	_InputStopController : MockPluginAutomationController(name := "InputController");
	_InputStopBranch : MockCompositeAutomationComponent(name := "InputBranch", parent := _InputStopController);

	_LifecycleLeaf : MockLeafAutomationComponent(name := "TestLeaf", parent := _TimeoutRoot);
	_EnableDisableLeaf : MockLeafAutomationComponent(name := "EnDisLeaf", parent := _TimeoutRoot);
	_IgnoreComposite : MockCompositeAutomationComponent(name := "CompIgnore", parent := _TimeoutRoot);
	_ContinueComposite : MockCompositeAutomationComponent(name := "CompContinue", parent := _TimeoutRoot);
	_StopComposite : MockCompositeAutomationComponent(name := "CompStop", parent := _TimeoutRoot);
	_BubbleComposite : MockCompositeAutomationComponent(name := "CompBubble", parent := _TimeoutRoot);
	_BubbleEvent : MockAutomationEvent(sourceObject := 0, eventId := 10, payload := "BubblePayload");
	_StopBubbleComposite : MockCompositeAutomationComponent(name := "CompStopBubble", parent := _TimeoutRoot);
	_StopBubbleEvent : MockAutomationEvent(sourceObject := 0, eventId := 20, payload := "StopPayload");
	_BroadcastComposite : MockCompositeAutomationComponent(name := "CompBcast", parent := _TimeoutRoot);
	_BroadcastEvent : MockAutomationEvent(sourceObject := 0, eventId := 30, payload := "BcastPayload");
	_InputOutputLeaf : MockLeafAutomationComponent(name := "IOLeaf", parent := _TimeoutRoot);
	_OutputPoliciesBranch : MockCompositeAutomationComponent(name := "OutputPolicies", parent := _TimeoutRoot);
	_InitializingProbeLeaf : MockLeafAutomationComponent(name := "InitProbe", parent := _TimeoutRoot);
	_WorkingProbeLeaf : MockLeafAutomationComponent(name := "WorkProbe", parent := _TimeoutRoot);
	_CallbackResetComposite : MockCompositeAutomationComponent(name := "CallbackReset", parent := _TimeoutRoot);
	_DuplicateBranch : MockCompositeAutomationComponent(name := "Duplicate", parent := _TimeoutRoot);
	_WrongParentBranch : MockCompositeAutomationComponent(name := "WrongParent", parent := _TimeoutRoot);
	_ForeignChildLeaf : MockLeafAutomationComponent(name := "Foreign", parent := _TimeoutRoot);

	_ResetPolicyLeaf : MockLeafAutomationComponent(name := "ResetPolicyLeaf", parent := _TimeoutRoot);
	_BeforeResetPolicyBranch : MockCompositeAutomationComponent(name := "BeforeResetPolicy", parent := _TimeoutRoot);
	_AfterResetPolicyBranch : MockCompositeAutomationComponent(name := "AfterResetPolicy", parent := _TimeoutRoot);
	_RecoverPolicyLeaf : MockLeafAutomationComponent(name := "RecoverPolicyLeaf", parent := _TimeoutRoot);
	_RecoverPolicyBranch : MockCompositeAutomationComponent(name := "RecoverPolicyBranch", parent := _TimeoutRoot);

	_AfterInitBranch : MockCompositeAutomationComponent(name := "AfterInitBranch", parent := _TimeoutRoot);
	_TimeoutNormLeaf : MockLeafAutomationComponent(name := "TimeoutNormLeaf", parent := _TimeoutRoot);

	_DisabledChildBranch : MockCompositeAutomationComponent(name := "DisabledChildBranch", parent := _TimeoutRoot);
	_CmdHmiPlugin : MockHmiControllerPlugin;
	_CmdHmiPlugins : ARRAY [0..0] OF TOF_Automation.IAutomationControllerPlugin := [_CmdHmiPlugin];
	_CmdHmiController : MockPluginAutomationController(name := "CmdHmiController");
END_VAR

(*!
<summary>Dispatches one scenario against the fresh fixture.</summary>
<description>Call once per fixture. Each method uses the assertions of the receiving case.</description>
<param name="scenario">Scenario assigned to the caller.</param>
<param name="assertions">Valid assertion context borrowed from the active case.</param>
*)
METHOD ExecuteScenario
VAR_INPUT
	scenario : AUTOMATION_COMPONENT_TEST_SCENARIO;
	assertions : REFERENCE TO TOF_Testing.Assertions;
END_VAR
CASE scenario OF
	AUTOMATION_COMPONENT_TEST_SCENARIO.LIFECYCLE_TRANSITIONS:
		testLifecycleTransitions(assertions := assertions);

	AUTOMATION_COMPONENT_TEST_SCENARIO.ENABLE_DISABLE:
		testEnableDisable(assertions := assertions);

	AUTOMATION_COMPONENT_TEST_SCENARIO.CHILD_ERROR_POLICY_IGNORE:
		testChildErrorPolicyIgnore(assertions := assertions);

	AUTOMATION_COMPONENT_TEST_SCENARIO.CHILD_ERROR_POLICY_SET_ERROR_AND_CONTINUE:
		testChildErrorPolicySetErrorAndContinue(assertions := assertions);

	AUTOMATION_COMPONENT_TEST_SCENARIO.CHILD_ERROR_POLICY_SET_ERROR_AND_STOP:
		testChildErrorPolicySetErrorAndStop(assertions := assertions);

	AUTOMATION_COMPONENT_TEST_SCENARIO.EVENT_BUBBLING:
		testEventBubbling(assertions := assertions);

	AUTOMATION_COMPONENT_TEST_SCENARIO.EVENT_BUBBLING_STOP_PROPAGATION:
		testEventBubblingStopPropagation(assertions := assertions);

	AUTOMATION_COMPONENT_TEST_SCENARIO.EVENT_BROADCASTING:
		testEventBroadcasting(assertions := assertions);

	AUTOMATION_COMPONENT_TEST_SCENARIO.INPUT_OUTPUT_PHASES:
		testInputOutputPhases(assertions := assertions);

	AUTOMATION_COMPONENT_TEST_SCENARIO.OUTPUT_PHASE_STOP:
		testOutputPhaseStop(assertions := assertions);

	AUTOMATION_COMPONENT_TEST_SCENARIO.INPUT_PHASE_STOP:
		testInputPhaseStop(assertions := assertions);

	AUTOMATION_COMPONENT_TEST_SCENARIO.OUTPUT_PHASE_CONTINUATION:
		testOutputPhaseContinuation(assertions := assertions);

	AUTOMATION_COMPONENT_TEST_SCENARIO.PRIMARY_ERROR_BEFORE_LOGGING:
		testPrimaryErrorBeforeLogging(assertions := assertions);

	AUTOMATION_COMPONENT_TEST_SCENARIO.RESET_CHILD_POLICIES:
		testResetChildPolicies(assertions := assertions);

	AUTOMATION_COMPONENT_TEST_SCENARIO.RESET_FROM_STOPPED_HOOK:
		testResetFromStoppedHook(assertions := assertions);

	AUTOMATION_COMPONENT_TEST_SCENARIO.PARENT_VALIDATION:
		testParentValidation(assertions := assertions);

	AUTOMATION_COMPONENT_TEST_SCENARIO.DUPLICATE_CHILD:
		testDuplicateChild(assertions := assertions);

	AUTOMATION_COMPONENT_TEST_SCENARIO.MISMATCHED_CHILD_PARENT:
		testMismatchedChildParent(assertions := assertions);

	AUTOMATION_COMPONENT_TEST_SCENARIO.INITIALIZATION_FAILURE_RESULT:
		testInitializationFailureResult(assertions := assertions);

	AUTOMATION_COMPONENT_TEST_SCENARIO.INDEXED_LOOKUP_CONTAINMENT:
		testIndexedLookupContainment(assertions := assertions);

	AUTOMATION_COMPONENT_TEST_SCENARIO.CONTROLLER_PLUGIN_RECOVERY:
		testControllerPluginRecovery(assertions := assertions);

	AUTOMATION_COMPONENT_TEST_SCENARIO.RESET_AND_RECOVER_IGNORE_EXCEPTION_POLICY:
		testResetAndRecoverIgnoreExceptionPolicy(assertions := assertions);

	AUTOMATION_COMPONENT_TEST_SCENARIO.AFTER_CHILDREN_INITIALIZING_AND_TIMEOUT_PROPAGATION:
		testAfterChildrenInitializingAndTimeoutPropagation(assertions := assertions);

	AUTOMATION_COMPONENT_TEST_SCENARIO.DISABLED_CHILD_STOP_RESET_AND_HMI_COMMAND_CONSUMPTION:
		testDisabledChildStopResetAndHmiCommandConsumption(assertions := assertions);
ELSE
	assertions.ThatBool(actual := FALSE, message := "Unknown automation component scenario").IsTrue();
END_CASE
END_METHOD

(*!
<summary>Borrows the concrete class name. Callers must not modify it.</summary>
*)
{attribute 'monitoring' := 'call'}
PROPERTY ClassName : REFERENCE TO STRING
GET
ClassName REF= _ClassName;
END_GET
END_PROPERTY

(*!
<summary>Borrows the project namespace name. Callers must not modify it.</summary>
*)
{attribute 'monitoring' := 'call'}
PROPERTY NamespaceName : REFERENCE TO STRING
GET
NamespaceName REF= CurrentNamespace.Name;
END_GET
END_PROPERTY

(*!
<summary>Checks continued child traversal with Ignore.</summary>
<description>
Uses the suite-owned root as the borrowed parent. Fixtures contain no cleanup-dependent local resources.
</description>
<param name="assertions">Valid assertion context borrowed from the active case.</param>
*)
METHOD PRIVATE testChildErrorPolicyIgnore
VAR_INPUT
	assertions : REFERENCE TO TOF_Testing.Assertions;
END_VAR
VAR
	i : INT;
END_VAR
_IgnoreComposite.Initialize();
_IgnoreComposite.ChildCriticalErrorHandlingPolicy := TOF_Automation.ChildCriticalErrorHandlingPolicies.Ignore;
_IgnoreComposite.ChildA.FailOnWorking := TRUE;

FOR i := 1 TO 3 DO
	_IgnoreComposite.Execute();
END_FOR

assertions.ThatDInt(
	actual := TO_DINT(_IgnoreComposite.ChildA.OperationalState),
	message := "ChildA should stop on critical error"
).ToBe(expected := TO_DINT(TOF_Automation.OPERATIONAL_STATE.STOPPED));

assertions.ThatDInt(
	actual := TO_DINT(_IgnoreComposite.OperationalState),
	message := "Composite should remain WORKING when policy is Ignore"
).ToBe(expected := TO_DINT(TOF_Automation.OPERATIONAL_STATE.WORKING));

assertions.ThatBool(
	actual := _IgnoreComposite.HasError,
	message := "Composite should not have error when policy is Ignore"
).IsFalse();

assertions.ThatInt(
	actual := _IgnoreComposite.ChildB.WorkingCount,
	message := "Later child must execute in every cycle with a retained critical sibling error"
).ToBe(expected := 3);
assertions.ThatInt(
	actual := _IgnoreComposite.AfterWorkingCount,
	message := "After-working hook must run after every continued traversal"
).ToBe(expected := 3);
END_METHOD

(*!
<summary>Checks continued child traversal with a copied noncritical error.</summary>
<description>
Uses the suite-owned root as the borrowed parent. Fixtures contain no cleanup-dependent local resources.
</description>
<param name="assertions">Valid assertion context borrowed from the active case.</param>
*)
METHOD PRIVATE testChildErrorPolicySetErrorAndContinue
VAR_INPUT
	assertions : REFERENCE TO TOF_Testing.Assertions;
END_VAR
VAR
	i : INT;
END_VAR
_ContinueComposite.Initialize();
_ContinueComposite.ChildCriticalErrorHandlingPolicy :=
	TOF_Automation.ChildCriticalErrorHandlingPolicies.SetErrorAndContinue;
_ContinueComposite.ChildA.FailOnWorking := TRUE;

FOR i := 1 TO 3 DO
	_ContinueComposite.Execute();
END_FOR

assertions.ThatBool(
	actual := _ContinueComposite.HasError,
	message := "Composite should record error when child fails with SetErrorAndContinue"
).IsTrue();

assertions.ThatDInt(
	actual := TO_DINT(_ContinueComposite.OperationalState),
	message := "Composite should remain WORKING when policy is SetErrorAndContinue"
).ToBe(expected := TO_DINT(TOF_Automation.OPERATIONAL_STATE.WORKING));

assertions.ThatInt(
	actual := _ContinueComposite.ChildB.WorkingCount,
	message := "Later child must execute in every cycle with a retained critical sibling error"
).ToBe(expected := 3);
assertions.ThatInt(
	actual := _ContinueComposite.AfterWorkingCount,
	message := "After-working hook must run after every continued traversal"
).ToBe(expected := 3);
assertions.ThatInt(
	actual := _ContinueComposite.RecoverCount,
	message := "Parent must not invoke OnRecover while faulted child remains critical"
).ToBe(expected := 0);

_ContinueComposite.ChildA.FailOnWorking := FALSE;
_ContinueComposite.ChildA.Reset();
_ContinueComposite.Execute();

assertions.ThatBool(
	actual := _ContinueComposite.HasError,
	message := "Parent should clear its copied error once the faulted child recovers"
).IsFalse();
assertions.ThatInt(
	actual := _ContinueComposite.RecoverCount,
	message := "Parent must invoke OnRecover once after the faulted child recovers"
).ToBe(expected := 1);
assertions.ThatInt(
	actual := _ContinueComposite.ChildA.WorkingCount,
	message := "Recovered child should resume working execution"
).ToBe(expected := 2);
END_METHOD

(*!
<summary>Checks stopping before later children after a critical child failure.</summary>
<description>
Uses the suite-owned root as the borrowed parent. Fixtures contain no cleanup-dependent local resources.
</description>
<param name="assertions">Valid assertion context borrowed from the active case.</param>
*)
METHOD PRIVATE testChildErrorPolicySetErrorAndStop
VAR_INPUT
	assertions : REFERENCE TO TOF_Testing.Assertions;
END_VAR
_StopComposite.Initialize();
_StopComposite.ChildCriticalErrorHandlingPolicy := TOF_Automation.ChildCriticalErrorHandlingPolicies.SetErrorAndStop;
_StopComposite.ChildA.FailOnWorking := TRUE;

_StopComposite.Execute();

assertions.ThatBool(
	actual := _StopComposite.HasError,
	message := "Composite should record error when child fails with SetErrorAndStop"
).IsTrue();

assertions.ThatDInt(
	actual := TO_DINT(_StopComposite.OperationalState),
	message := "Composite should transition to STOPPED when policy is SetErrorAndStop"
).ToBe(expected := TO_DINT(TOF_Automation.OPERATIONAL_STATE.STOPPED));

assertions.ThatInt(
	actual := _StopComposite.ChildB.WorkingCount,
	message := "Stop policy must not execute later children"
).ToBe(expected := 0);
assertions.ThatInt(
	actual := _StopComposite.AfterWorkingCount,
	message := "Stop policy must not complete the working phase"
).ToBe(expected := 0);
END_METHOD

(*!
<summary>Checks leaf enablement with a live parent.</summary>
<description>
Uses the suite-owned root as the borrowed parent. Fixtures contain no cleanup-dependent local resources.
</description>
<param name="assertions">Valid assertion context borrowed from the active case.</param>
*)
METHOD PRIVATE testEnableDisable
VAR_INPUT
	assertions : REFERENCE TO TOF_Testing.Assertions;
END_VAR
_EnableDisableLeaf.Initialize();

_EnableDisableLeaf.Disable();
assertions.ThatBool(actual := _EnableDisableLeaf.Enabled, message := "Leaf should be disabled").IsFalse();
assertions.ThatInt(
	actual := _EnableDisableLeaf.DisableCount,
	message := "DisableCount should be 1"
).ToBe(expected := 1);

_EnableDisableLeaf.Execute();
assertions.ThatInt(
	actual := _EnableDisableLeaf.WorkingCount,
	message := "Disabled leaf must not execute OnWorking"
).ToBe(expected := 0);

_EnableDisableLeaf.Enable(includeChildren := TRUE);
assertions.ThatBool(actual := _EnableDisableLeaf.Enabled, message := "Leaf should be enabled").IsTrue();
assertions.ThatInt(
	actual := _EnableDisableLeaf.EnableCount,
	message := "EnableCount should be 1"
).ToBe(expected := 1);

_EnableDisableLeaf.Execute();
assertions.ThatInt(
	actual := _EnableDisableLeaf.WorkingCount,
	message := "Enabled leaf should execute OnWorking"
).ToBe(expected := 1);
END_METHOD

(*!
<summary>Checks broadcast delivery to two children.</summary>
<description>
Uses the suite-owned root as the borrowed parent. Fixtures contain no cleanup-dependent local resources.
</description>
<param name="assertions">Valid assertion context borrowed from the active case.</param>
*)
METHOD PRIVATE testEventBroadcasting
VAR_INPUT
	assertions : REFERENCE TO TOF_Testing.Assertions;
END_VAR
_BroadcastComposite.BroadcastEvent(event := _BroadcastEvent);

assertions.ThatInt(
	actual := _BroadcastComposite.ChildA.LastReceivedEventId,
	message := "ChildA should receive broadcast event"
).ToBe(expected := 30);

assertions.ThatInt(
	actual := _BroadcastComposite.ChildB.LastReceivedEventId,
	message := "ChildB should receive broadcast event"
).ToBe(expected := 30);
END_METHOD

(*!
<summary>Checks event bubbling through a live parent.</summary>
<description>
Uses the suite-owned root as the borrowed parent. Fixtures contain no cleanup-dependent local resources.
</description>
<param name="assertions">Valid assertion context borrowed from the active case.</param>
*)
METHOD PRIVATE testEventBubbling
VAR_INPUT
	assertions : REFERENCE TO TOF_Testing.Assertions;
END_VAR
_BubbleComposite.ChildA.BubbleEvent(event := _BubbleEvent);

assertions.ThatInt(
	actual := _BubbleComposite.ChildA.LastReceivedEventId,
	message := "ChildA should receive event locally"
).ToBe(expected := 10);

assertions.ThatInt(
	actual := _BubbleComposite.LastReceivedEventId,
	message := "Parent composite should receive bubbled event"
).ToBe(expected := 10);
END_METHOD

(*!
<summary>Checks local bubbling termination.</summary>
<description>
Uses the suite-owned root as the borrowed parent. Fixtures contain no cleanup-dependent local resources.
</description>
<param name="assertions">Valid assertion context borrowed from the active case.</param>
*)
METHOD PRIVATE testEventBubblingStopPropagation
VAR_INPUT
	assertions : REFERENCE TO TOF_Testing.Assertions;
END_VAR
_StopBubbleComposite.ChildA.StopPropagationOnEvent := TRUE;
_StopBubbleComposite.ChildA.BubbleEvent(event := _StopBubbleEvent);

assertions.ThatInt(
	actual := _StopBubbleComposite.ChildA.LastReceivedEventId,
	message := "ChildA should receive event locally"
).ToBe(expected := 20);

assertions.ThatInt(
	actual := _StopBubbleComposite.EventReceivedCount,
	message := "Parent composite must not receive event when propagation stopped"
).ToBe(expected := 0);
END_METHOD

(*!
<summary>Checks direct leaf input, work and output calls.</summary>
<description>
Uses the suite-owned root as the borrowed parent. Fixtures contain no cleanup-dependent local resources.
</description>
<param name="assertions">Valid assertion context borrowed from the active case.</param>
*)
METHOD PRIVATE testInputOutputPhases
VAR_INPUT
	assertions : REFERENCE TO TOF_Testing.Assertions;
END_VAR
_InputOutputLeaf.Initialize();

_InputOutputLeaf.ProcessInput();
assertions.ThatInt(
	actual := _InputOutputLeaf.ProcessInputCount,
	message := "ProcessInputCount should be 1"
).ToBe(expected := 1);

_InputOutputLeaf.Execute();
assertions.ThatInt(
	actual := _InputOutputLeaf.WorkingCount,
	message := "WorkingCount should be 1"
).ToBe(expected := 1);

_InputOutputLeaf.ProcessOutput();
assertions.ThatInt(
	actual := _InputOutputLeaf.ProcessOutputCount,
	message := "ProcessOutputCount should be 1"
).ToBe(expected := 1);
END_METHOD

(*!
<summary>Checks leaf lifecycle transitions with a live parent.</summary>
<description>
Uses the suite-owned root as the borrowed parent. Fixtures contain no cleanup-dependent local resources.
</description>
<param name="assertions">Valid assertion context borrowed from the active case.</param>
*)
METHOD PRIVATE testLifecycleTransitions
VAR_INPUT
	assertions : REFERENCE TO TOF_Testing.Assertions;
END_VAR
assertions.ThatDInt(
	actual := TO_DINT(_LifecycleLeaf.OperationalState),
	message := "Initial state should be INITIALIZING"
).ToBe(expected := TO_DINT(TOF_Automation.OPERATIONAL_STATE.INITIALIZING));

_LifecycleLeaf.Initialize();
assertions.ThatDInt(
	actual := TO_DINT(_LifecycleLeaf.OperationalState),
	message := "State should be WORKING after Initialize"
).ToBe(expected := TO_DINT(TOF_Automation.OPERATIONAL_STATE.WORKING));

_LifecycleLeaf.Execute();
assertions.ThatInt(actual := _LifecycleLeaf.WorkingCount, message := "WorkingCount should be 1").ToBe(expected := 1);

_LifecycleLeaf.Stop(reason := "Manual test stop");
assertions.ThatDInt(
	actual := TO_DINT(_LifecycleLeaf.OperationalState),
	message := "State should be STOPPED after Stop"
).ToBe(expected := TO_DINT(TOF_Automation.OPERATIONAL_STATE.STOPPED));
assertions.ThatWideString(
	actual := _LifecycleLeaf.OperationalStateReason,
	message := "OperationalStateReason should match stop reason"
).ToBe(expected := "Manual test stop");

_LifecycleLeaf.Reset();
assertions.ThatDInt(
	actual := TO_DINT(_LifecycleLeaf.OperationalState),
	message := "State should return to WORKING after Reset"
).ToBe(expected := TO_DINT(TOF_Automation.OPERATIONAL_STATE.WORKING));
END_METHOD

(*!
<summary>Checks reset traversal and parent recovery for all three critical-child policies.</summary>
<description>
Runs once on a fresh fixture. Borrowed objects remain live for the call.
</description>
<param name="assertions">Valid assertion context borrowed from the active case.</param>
*)
METHOD PRIVATE testResetChildPolicies
VAR_INPUT
	assertions : REFERENCE TO TOF_Testing.Assertions;
END_VAR
_ResetIgnoreBranch.Initialize();
_ResetContinueBranch.Initialize();
_ResetStopBranch.Initialize();
_ResetIgnoreBranch.Stop(reason := "Reset regression");
_ResetContinueBranch.Stop(reason := "Reset regression");
_ResetStopBranch.Stop(reason := "Reset regression");
_ResetIgnoreBranch.ChildCriticalErrorHandlingPolicy := TOF_Automation.ChildCriticalErrorHandlingPolicies.Ignore;
_ResetContinueBranch.ChildCriticalErrorHandlingPolicy :=
	TOF_Automation.ChildCriticalErrorHandlingPolicies.SetErrorAndContinue;
_ResetStopBranch.ChildCriticalErrorHandlingPolicy := TOF_Automation.ChildCriticalErrorHandlingPolicies.SetErrorAndStop;
_ResetIgnoreBranch.ChildA.ThrowOnReset := TRUE;
_ResetContinueBranch.ChildA.ThrowOnReset := TRUE;
_ResetStopBranch.ChildA.ThrowOnReset := TRUE;

_ResetIgnoreBranch.Reset();
_ResetContinueBranch.Reset();
_ResetStopBranch.Reset();

assertions.ThatDInt(
	actual := TO_DINT(_ResetIgnoreBranch.OperationalState),
	message := "Ignore resumes parent despite stopped child"
).ToBe(expected := TO_DINT(TOF_Automation.OPERATIONAL_STATE.WORKING));
assertions.ThatDInt(
	actual := TO_DINT(_ResetContinueBranch.OperationalState),
	message := "Continue resumes parent despite stopped child"
).ToBe(expected := TO_DINT(TOF_Automation.OPERATIONAL_STATE.WORKING));
assertions.ThatDInt(
	actual := TO_DINT(_ResetStopBranch.OperationalState),
	message := "Stop refuses parent recovery"
).ToBe(expected := TO_DINT(TOF_Automation.OPERATIONAL_STATE.STOPPED));
assertions.ThatInt(
	actual := _ResetIgnoreBranch.ChildB.ResetCount,
	message := "Ignore resets later child"
).ToBe(expected := 1);
assertions.ThatInt(
	actual := _ResetContinueBranch.ChildB.ResetCount,
	message := "Continue resets later child"
).ToBe(expected := 1);
assertions.ThatInt(
	actual := _ResetStopBranch.ChildB.ResetCount,
	message := "Stop ends reset traversal"
).ToBe(expected := 0);
assertions.ThatBool(
	actual := _ResetIgnoreBranch.HasError,
	message := "Ignore leaves the child diagnostic local"
).IsFalse();
assertions.ThatBool(
	actual := _ResetContinueBranch.HasError,
	message := "Continue retains the child diagnostic"
).IsTrue();
assertions.ThatDInt(
	actual := TO_DINT(_ResetContinueBranch.Error.Severity),
	message := "Continue downgrades copied severity"
).ToBe(expected := TO_DINT(TOF_Core.ERROR_SEVERITY.ERROR));
assertions.ThatBool(actual := _ResetStopBranch.HasError, message := "Stop records critical child failure").IsTrue();
assertions.ThatDInt(
	actual := TO_DINT(_ResetIgnoreBranch.ChildA.OperationalState),
	message := "Failed child stays stopped"
).ToBe(expected := TO_DINT(TOF_Automation.OPERATIONAL_STATE.STOPPED));
assertions.ThatDInt(
	actual := TO_DINT(_ResetContinueBranch.ChildA.OperationalState),
	message := "Continue does not revive failed child"
).ToBe(expected := TO_DINT(TOF_Automation.OPERATIONAL_STATE.STOPPED));
END_METHOD

(*!
<summary>Checks that reset from a stopped hook is not undone by the current traversal.</summary>
<description>
Runs once on a fresh fixture. Borrowed objects remain live for the call.
</description>
<param name="assertions">Valid assertion context borrowed from the active case.</param>
*)
METHOD PRIVATE testResetFromStoppedHook
VAR_INPUT
	assertions : REFERENCE TO TOF_Testing.Assertions;
END_VAR
_CallbackResetComposite.Initialize();
_CallbackResetComposite.Stop(reason := "Callback reset regression");
_CallbackResetComposite.ResetOnBeforeChildrenStopped := TRUE;
_CallbackResetComposite.Execute();

assertions.ThatDInt(
	actual := TO_DINT(_CallbackResetComposite.OperationalState),
	message := "Callback reset resumes the parent"
).ToBe(expected := TO_DINT(TOF_Automation.OPERATIONAL_STATE.WORKING));
assertions.ThatDInt(
	actual := TO_DINT(_CallbackResetComposite.ChildA.OperationalState),
	message := "Current doStop must not stop reset ChildA"
).ToBe(expected := TO_DINT(TOF_Automation.OPERATIONAL_STATE.WORKING));
assertions.ThatDInt(
	actual := TO_DINT(_CallbackResetComposite.ChildB.OperationalState),
	message := "Current doStop must not stop reset ChildB"
).ToBe(expected := TO_DINT(TOF_Automation.OPERATIONAL_STATE.WORKING));
assertions.ThatInt(
	actual := _CallbackResetComposite.ChildA.WorkingCount,
	message := "Recovery does not restart working traversal within the stopped phase"
).ToBe(expected := 0);

_CallbackResetComposite.Execute();

assertions.ThatInt(
	actual := _CallbackResetComposite.ChildA.WorkingCount,
	message := "ChildA works next cycle"
).ToBe(expected := 1);
assertions.ThatInt(
	actual := _CallbackResetComposite.ChildB.WorkingCount,
	message := "ChildB works next cycle"
).ToBe(expected := 1);
assertions.ThatInt(
	actual := _CallbackResetComposite.AfterWorkingCount,
	message := "Working traversal completes"
).ToBe(expected := 1);
END_METHOD

(*!
<summary>Checks parent rejection before ready and pending initialization hooks.</summary>
<description>
Runs once on a fresh fixture. Borrowed objects remain live for the call.
</description>
<param name="assertions">Valid assertion context borrowed from the active case.</param>
*)
METHOD PRIVATE testParentValidation
VAR_INPUT
	assertions : REFERENCE TO TOF_Testing.Assertions;
END_VAR
VAR
	initialized : BOOL;
END_VAR
_OrphanPendingLeaf.InitReturnValue := FALSE;
_OrphanPendingBranch.ChildA.InitReturnValue := FALSE;
_ValidPendingLeaf.InitReturnValue := FALSE;

initialized := _OrphanReadyLeaf.Initialize();
assertions.ThatBool(actual := initialized, message := "Ready orphan leaf must fail").IsFalse();
initialized := _OrphanPendingLeaf.Initialize();
assertions.ThatBool(actual := initialized, message := "Pending orphan leaf must fail").IsFalse();
initialized := _OrphanReadyBranch.Initialize();
assertions.ThatBool(actual := initialized, message := "Ready orphan branch must fail").IsFalse();
initialized := _OrphanPendingBranch.Initialize();
assertions.ThatBool(actual := initialized, message := "Pending orphan branch must fail").IsFalse();
assertions.ThatInt(
	actual := _OrphanReadyLeaf.InitializeCount,
	message := "Ready leaf hook must not run"
).ToBe(expected := 0);
assertions.ThatInt(
	actual := _OrphanPendingLeaf.InitializeCount,
	message := "Pending leaf hook must not run"
).ToBe(expected := 0);
assertions.ThatInt(
	actual := _OrphanReadyBranch.BeforeInitializeCount,
	message := "Ready branch hook must not run"
).ToBe(expected := 0);
assertions.ThatInt(
	actual := _OrphanPendingBranch.BeforeInitializeCount,
	message := "Pending branch hook must not run"
).ToBe(expected := 0);
assertions.ThatDInt(
	actual := TO_DINT(_OrphanReadyLeaf.OperationalState),
	message := "Orphan leaf is terminal INVALID"
).ToBe(expected := TO_DINT(TOF_Automation.OPERATIONAL_STATE.INVALID));
assertions.ThatDInt(
	actual := TO_DINT(_OrphanReadyBranch.OperationalState),
	message := "Orphan branch is terminal INVALID"
).ToBe(expected := TO_DINT(TOF_Automation.OPERATIONAL_STATE.INVALID));
assertions.ThatBool(
	actual := _OrphanPendingLeaf.HasError,
	message := "Missing parent produces a copied error"
).IsTrue();
assertions.ThatBool(
	actual := _OrphanPendingBranch.HasError,
	message := "Missing parent produces a branch error"
).IsTrue();

initialized := _ValidPendingLeaf.Initialize();
assertions.ThatBool(actual := initialized, message := "Valid pending leaf reports incomplete work").IsFalse();
assertions.ThatDInt(
	actual := TO_DINT(_ValidPendingLeaf.OperationalState),
	message := "Valid pending leaf remains initializing"
).ToBe(expected := TO_DINT(TOF_Automation.OPERATIONAL_STATE.INITIALIZING));
assertions.ThatInt(
	actual := _ValidPendingLeaf.InitializeCount,
	message := "Valid leaf hook is invoked"
).ToBe(expected := 1);
_ValidPendingLeaf.InitReturnValue := TRUE;
initialized := _ValidPendingLeaf.Initialize();
assertions.ThatBool(actual := initialized, message := "Valid leaf can finish initialization").IsTrue();
initialized := _EmptyRoot.Initialize();
assertions.ThatBool(actual := initialized, message := "Empty root composition is valid").IsTrue();
END_METHOD

(*!
<summary>Checks failure results, preflight and propagation through two branch levels.</summary>
<description>
Runs once on a fresh fixture. Borrowed objects remain live for the call.
</description>
<param name="assertions">Valid assertion context borrowed from the active case.</param>
*)
METHOD PRIVATE testInitializationFailureResult
VAR_INPUT
	assertions : REFERENCE TO TOF_Testing.Assertions;
END_VAR
VAR
	initialized : BOOL;
END_VAR
_FirstNullBranch.Children[0] := 0;
_SecondNullBranch.Children[1] := 0;
_ThrowingChildBranch.ChildA.ThrowOnInitializing := TRUE;
_FailureOuterBranch.Children[0] := _FailureInnerBranch;
_FailureInnerBranch.Children[1] := 0;

initialized := _FirstNullBranch.Initialize();
assertions.ThatBool(actual := initialized, message := "First null slot must not return success").IsFalse();
initialized := _SecondNullBranch.Initialize();
assertions.ThatBool(actual := initialized, message := "Later null slot must not return success").IsFalse();
assertions.ThatInt(
	actual := _FirstNullBranch.BeforeInitializeCount,
	message := "Null slot rejection precedes branch callbacks"
).ToBe(expected := 0);
assertions.ThatInt(
	actual := _SecondNullBranch.ChildA.InitializeCount,
	message := "Later null slot rejection precedes earlier child callbacks"
).ToBe(expected := 0);
initialized := _ThrowingChildBranch.Initialize();
assertions.ThatBool(
	actual := initialized,
	message := "Failed child initialization must not return success"
).IsFalse();
assertions.ThatDInt(
	actual := TO_DINT(_ThrowingChildBranch.OperationalState),
	message := "Parent immediately propagates INVALID child"
).ToBe(expected := TO_DINT(TOF_Automation.OPERATIONAL_STATE.INVALID));
assertions.ThatInt(
	actual := _ThrowingChildBranch.ChildB.InitializeCount,
	message := "No later child initializes after a terminal child failure"
).ToBe(expected := 0);
assertions.ThatBool(
	actual := _ThrowingChildBranch.HasError,
	message := "Child failure is copied to parent"
).IsTrue();
initialized := _FailureOuterBranch.Initialize();
assertions.ThatBool(actual := initialized, message := "Nested invalid branch must not appear ready").IsFalse();
assertions.ThatDInt(
	actual := TO_DINT(_FailureInnerBranch.OperationalState),
	message := "Inner branch is INVALID"
).ToBe(expected := TO_DINT(TOF_Automation.OPERATIONAL_STATE.INVALID));
assertions.ThatDInt(
	actual := TO_DINT(_FailureOuterBranch.OperationalState),
	message := "Outer branch immediately becomes INVALID"
).ToBe(expected := TO_DINT(TOF_Automation.OPERATIONAL_STATE.INVALID));
assertions.ThatBool(actual := _FailureOuterBranch.HasError, message := "Nested error survives propagation").IsTrue();
END_METHOD

(*!
<summary>Checks borrowed lookup identity, bounds and throwing or missing storage.</summary>
<description>
Catches unexpected escapes into an explicit test failure. Terminal OOM is excluded from this shared
suite and is verified separately in an isolated application. No fixture owns cleanup-dependent resources.
</description>
<param name="assertions">Valid assertion context borrowed from the active case.</param>
*)
METHOD PRIVATE testIndexedLookupContainment
VAR_INPUT
	assertions : REFERENCE TO TOF_Testing.Assertions;
END_VAR
VAR
	expected : TOF_Automation.IChildAutomationComponent;
	actual : TOF_Automation.IChildAutomationComponent;
	exceptionEscaped : BOOL;
	exceptionCode : __SYSTEM.ExceptionCode;
END_VAR
__TRY
	expected := _LookupComposite.ChildA;
	actual := _LookupComposite.TryGetChildByIndex(index := 0);
	assertions.ThatBool(actual := actual = expected, message := "Composite lookup returns the borrowed child").IsTrue();
	actual := _LookupComposite.TryGetChildByIndex(index := 2);
	assertions.ThatBool(actual := actual = 0, message := "Out-of-range lookup returns null").IsTrue();
	_LookupComposite.ThrowOnGetChildren := TRUE;
	actual := _LookupComposite.TryGetChildByIndex(index := 0);
	assertions.ThatBool(actual := actual = 0, message := "Composite getter exception is contained").IsTrue();
	_LookupComposite.ThrowOnGetChildren := FALSE;
	_LookupComposite.MissingChildrenReference := TRUE;
	actual := _LookupComposite.TryGetChildByIndex(index := 0);
	assertions.ThatBool(actual := actual = 0, message := "Missing composite storage returns null").IsTrue();
	expected := _LookupController.Child;
	actual := _LookupController.TryGetChildByIndex(index := 0);
	assertions.ThatBool(actual := actual = expected, message := "Controller lookup returns borrowed child").IsTrue();
	_LookupController.ThrowOnGetChildren := TRUE;
	actual := _LookupController.TryGetChildByIndex(index := 0);
	assertions.ThatBool(actual := actual = 0, message := "Controller getter exception is contained").IsTrue();
	_LookupController.ThrowOnGetChildren := FALSE;
	_LookupController.MissingChildrenReference := TRUE;
	actual := _LookupController.TryGetChildByIndex(index := 0);
	assertions.ThatBool(actual := actual = 0, message := "Missing controller storage returns null").IsTrue();
__CATCH(exceptionCode)
	exceptionEscaped := TRUE;
__ENDTRY

assertions.ThatBool(
	actual := exceptionEscaped,
	message := "No exception may escape an indexed Try lookup"
).IsFalse();
END_METHOD

(*!
<summary>Checks disabled HMI service, same-cycle guards and stopped-tree reset.</summary>
<description>
Uses real base HMI command/status methods. An injected failure while disabled must require Reset.
All borrowed fixtures remain live for the call; no cleanup-dependent resources are owned locally.
</description>
<param name="assertions">Valid assertion context borrowed from the active case.</param>
*)
METHOD PRIVATE testControllerPluginRecovery
VAR_INPUT
	assertions : REFERENCE TO TOF_Testing.Assertions;
END_VAR
VAR
	actualPlugin : TOF_Automation.IAutomationControllerPlugin;
	expectedPlugin : TOF_Automation.IAutomationControllerPlugin;
END_VAR
_HmiController.ConfigurePlugins(plugins := _HmiPlugins);
_HmiController.Execute();
assertions.ThatInt(
	actual := _HmiPlugin.BeforeCount,
	message := "Initializing root has no plugin service"
).ToBe(expected := 0);
_HmiController.Initialize();
expectedPlugin := _HmiPlugin;
actualPlugin := _HmiController.TryGetPluginByIndex(index := 0);
assertions.ThatBool(
	actual := actualPlugin = expectedPlugin,
	message := "Plugin lookup preserves borrowed identity"
).IsTrue();
actualPlugin := _HmiController.TryGetPluginByIndex(index := 1);
assertions.ThatBool(actual := actualPlugin = 0, message := "Missing plugin index returns null").IsTrue();
_HmiPlugin.AutomationComponentCommands.Disable := TRUE;
_HmiController.Execute();

assertions.ThatBool(actual := _HmiController.Enabled, message := "HMI Disable reaches the root").IsFalse();
assertions.ThatBool(
	actual := _HmiPlugin.AutomationComponentCommands.Disable,
	message := "Disable command is consumed"
).IsFalse();
assertions.ThatBool(
	actual := _HmiPlugin.AutomationComponentStatuses.Enabled,
	message := "Disabled status is refreshed"
).IsFalse();
assertions.ThatInt(
	actual := _HmiController.Child.ProcessInputCount,
	message := "Disable skips same-cycle input"
).ToBe(expected := 0);
assertions.ThatInt(
	actual := _HmiController.Child.WorkingCount,
	message := "Disable skips same-cycle work"
).ToBe(expected := 0);
assertions.ThatInt(
	actual := _HmiController.Child.ProcessOutputCount,
	message := "Disable skips same-cycle output"
).ToBe(expected := 0);
_HmiController.Execute();
assertions.ThatInt(
	actual := _HmiPlugin.BeforeCount,
	message := "Disabled root keeps before service"
).ToBe(expected := 2);
assertions.ThatInt(
	actual := _HmiPlugin.AfterCount,
	message := "Disabled root keeps after service"
).ToBe(expected := 2);
assertions.ThatInt(
	actual := _HmiController.Child.WorkingCount,
	message := "Disabled interval has no work"
).ToBe(expected := 0);
_HmiPlugin.AutomationComponentCommands.Enable := TRUE;
_HmiController.Execute();

assertions.ThatBool(actual := _HmiController.Enabled, message := "The same HMI channel can re-enable root").IsTrue();
assertions.ThatBool(
	actual := _HmiPlugin.AutomationComponentStatuses.Enabled,
	message := "Enabled status is refreshed"
).IsTrue();
assertions.ThatBool(
	actual := _HmiPlugin.AutomationComponentCommands.Enable,
	message := "Enable command is consumed"
).IsFalse();
assertions.ThatInt(
	actual := _HmiController.Child.ProcessInputCount,
	message := "Input resumes on Enable"
).ToBe(expected := 1);
assertions.ThatInt(
	actual := _HmiController.Child.WorkingCount,
	message := "Work resumes on Enable"
).ToBe(expected := 1);
assertions.ThatInt(
	actual := _HmiController.Child.ProcessOutputCount,
	message := "Output resumes on Enable"
).ToBe(expected := 1);
_HmiController.Stop(reason := "HMI stopped recovery regression");
_HmiController.Execute();
assertions.ThatInt(
	actual := _HmiController.Child.StopCount,
	message := "Enabled stopped hooks still run"
).ToBe(expected := 1);
assertions.ThatInt(
	actual := _HmiController.Child.ProcessInputCount,
	message := "Stopped root retains input"
).ToBe(expected := 2);
assertions.ThatInt(
	actual := _HmiController.Child.ProcessOutputCount,
	message := "Stopped root retains output"
).ToBe(expected := 2);
_HmiPlugin.AutomationComponentCommands.Reset := TRUE;
_HmiController.Execute();
assertions.ThatDInt(
	actual := TO_DINT(_HmiController.OperationalState),
	message := "HMI Reset resumes root"
).ToBe(expected := TO_DINT(TOF_Automation.OPERATIONAL_STATE.WORKING));
assertions.ThatInt(
	actual := _HmiController.Child.WorkingCount,
	message := "HMI Reset resumes child work"
).ToBe(expected := 2);
assertions.ThatInt(
	actual := _HmiPlugin.AfterCount,
	message := "Every managed cycle refreshes status"
).ToBe(expected := 5);

_HmiPlugin.AutomationComponentCommands.Disable := TRUE;
_HmiController.Execute();
_HmiPlugin.ThrowOnBeforeExecute := TRUE;
_HmiController.Execute();
assertions.ThatDInt(
	actual := TO_DINT(_HmiController.OperationalState),
	message := "Failed disabled service must require Reset"
).ToBe(expected := TO_DINT(TOF_Automation.OPERATIONAL_STATE.STOPPED));
assertions.ThatBool(
	actual := _HmiController.HasError,
	message := "Disabled plugin failure retains its copied error"
).IsTrue();
assertions.ThatInt(
	actual := _HmiController.Child.WorkingCount,
	message := "Disabled fault does no work"
).ToBe(expected := 2);
_HmiPlugin.ThrowOnBeforeExecute := FALSE;
_HmiPlugin.AutomationComponentCommands.Enable := TRUE;
_HmiPlugin.AutomationComponentCommands.Reset := TRUE;
_HmiController.Execute();
assertions.ThatBool(
	actual := _HmiController.HasError,
	message := "Explicit recovery clears the plugin failure"
).IsFalse();
assertions.ThatBool(
	actual := _HmiPlugin.AutomationComponentCommands.Reset,
	message := "Recovery Reset is consumed"
).IsFalse();
assertions.ThatInt(
	actual := _HmiController.Child.WorkingCount,
	message := "Enable and Reset resume work"
).ToBe(expected := 3);

_InvalidHmiController.ConfigurePlugins(plugins := _HmiPlugins);
_InvalidHmiController.MissingChildrenReference := TRUE;
_InvalidHmiController.Initialize();
_InvalidHmiController.Execute();
assertions.ThatInt(
	actual := _HmiPlugin.BeforeCount,
	message := "INVALID root has no before service"
).ToBe(expected := 8);
assertions.ThatInt(
	actual := _HmiPlugin.AfterCount,
	message := "INVALID root has no after service"
).ToBe(expected := 8);
END_METHOD

(*!
<summary>Checks that a duplicate child invalidates a branch before initialization callbacks.</summary>
<param name="assertions">Valid assertion context borrowed from the active case.</param>
*)
METHOD PRIVATE testDuplicateChild
VAR_INPUT
	assertions : REFERENCE TO TOF_Testing.Assertions;
END_VAR
_DuplicateBranch.Children[1] := _DuplicateBranch.Children[0];
_DuplicateBranch.ChildCriticalErrorHandlingPolicy := TOF_Automation.ChildCriticalErrorHandlingPolicies.Ignore;

assertions.ThatBool(actual := _DuplicateBranch.Initialize(), message := "Invalid composition must fail").IsFalse();
assertions.ThatBool(
	actual := _DuplicateBranch.OperationalState = TOF_Automation.OPERATIONAL_STATE.INVALID,
	message := "Branch must enter INVALID"
).IsTrue();
assertions.ThatBool(
	actual := _DuplicateBranch.HasError AND_THEN _DuplicateBranch.Error.Severity = TOF_Core.ERROR_SEVERITY.CRITICAL,
	message := "Branch must retain a critical error"
).IsTrue();
assertions.ThatWideString(
	actual := _DuplicateBranch.OperationalStateReason,
	message := "Diagnosis identifies the conflicting slots"
).ToBe(expected := "Duplicate: Children[1] (ChildA) duplicates Children[0]");
assertions.ThatInt(
	actual := _DuplicateBranch.BeforeInitializeCount,
	message := "Branch hook must not run"
).ToBe(expected := 0);
assertions.ThatInt(
	actual := _DuplicateBranch.ChildA.InitializeCount,
	message := "First child must not start"
).ToBe(expected := 0);
assertions.ThatBool(
	actual := _DuplicateBranch.Initialize(),
	message := "Invalid branch must remain terminal"
).IsFalse();
END_METHOD

(*!
<summary>Checks that a mismatched parent invalidates a branch before initialization callbacks.</summary>
<param name="assertions">Valid assertion context borrowed from the active case.</param>
*)
METHOD PRIVATE testMismatchedChildParent
VAR_INPUT
	assertions : REFERENCE TO TOF_Testing.Assertions;
END_VAR
_WrongParentBranch.Children[1] := _ForeignChildLeaf;
_WrongParentBranch.ChildCriticalErrorHandlingPolicy := TOF_Automation.ChildCriticalErrorHandlingPolicies.Ignore;

assertions.ThatBool(actual := _WrongParentBranch.Initialize(), message := "Invalid composition must fail").IsFalse();
assertions.ThatBool(
	actual := _WrongParentBranch.OperationalState = TOF_Automation.OPERATIONAL_STATE.INVALID,
	message := "Branch must enter INVALID"
).IsTrue();
assertions.ThatBool(
	actual := _WrongParentBranch.HasError
		AND_THEN _WrongParentBranch.Error.Severity = TOF_Core.ERROR_SEVERITY.CRITICAL,
	message := "Branch must retain a critical error"
).IsTrue();
assertions.ThatWideString(
	actual := _WrongParentBranch.OperationalStateReason,
	message := "Diagnosis identifies the conflicting slot"
).ToBe(expected := "WrongParent: Children[1] (Foreign) has a different Parent");
assertions.ThatInt(
	actual := _WrongParentBranch.BeforeInitializeCount,
	message := "Branch hook must not run"
).ToBe(expected := 0);
assertions.ThatInt(
	actual := _WrongParentBranch.ChildA.InitializeCount,
	message := "First child must not start"
).ToBe(expected := 0);
assertions.ThatBool(
	actual := _WrongParentBranch.Initialize(),
	message := "Invalid branch must remain terminal"
).IsFalse();
END_METHOD

(*!
<summary>Checks interrupted controller and composite output passes and the following stopped pass.</summary>
<param name="assertions">Valid assertion context borrowed from the active case.</param>
*)
METHOD PRIVATE testOutputPhaseStop
VAR_INPUT
	assertions : REFERENCE TO TOF_Testing.Assertions;
END_VAR
_OutputStopBranch.Initialize();
_OutputStopBranch.ChildCriticalErrorHandlingPolicy :=
	TOF_Automation.ChildCriticalErrorHandlingPolicies.SetErrorAndStop;
_OutputStopBranch.ChildA.ThrowOnNextOutput := TRUE;
_OutputStopBranch.ProcessOutput();
assertions.ThatBool(
	actual := _OutputStopBranch.OperationalState = TOF_Automation.OPERATIONAL_STATE.STOPPED,
	message := "Branch stops"
).IsTrue();
assertions.ThatInt(
	actual := _OutputStopBranch.ChildA.ProcessOutputCount,
	message := "First output already ran"
).ToBe(expected := 1);
assertions.ThatInt(
	actual := _OutputStopBranch.ChildB.ProcessOutputCount,
	message := "Later output is deferred"
).ToBe(expected := 0);
assertions.ThatInt(
	actual := _OutputStopBranch.AfterOutputCount,
	message := "Interrupted branch skips after hook"
).ToBe(expected := 0);

_OutputStopBranch.ProcessOutput();
assertions.ThatInt(
	actual := _OutputStopBranch.ChildA.ProcessOutputCount,
	message := "Stopped pass starts at slot 0"
).ToBe(expected := 2);
assertions.ThatInt(
	actual := _OutputStopBranch.ChildB.ProcessOutputCount,
	message := "Stopped pass reaches slot 1"
).ToBe(expected := 1);
assertions.ThatInt(
	actual := _OutputStopBranch.AfterOutputCount,
	message := "Stopped pass completes"
).ToBe(expected := 1);

_OutputStopController.Initialize();
_OutputStopController.ChildCriticalErrorHandlingPolicy :=
	TOF_Automation.ChildCriticalErrorHandlingPolicies.SetErrorAndStop;
_OutputStopController.Child.ThrowOnNextOutput := TRUE;
_OutputStopController.Execute();
assertions.ThatInt(
	actual := _OutputStopController.Child.ProcessOutputCount,
	message := "Controller output ran"
).ToBe(expected := 1);
assertions.ThatInt(
	actual := _OutputStopController.AfterOutputCount,
	message := "Interrupted last slot skips hook"
).ToBe(expected := 0);

_OutputStopController.Execute();
assertions.ThatInt(
	actual := _OutputStopController.Child.ProcessOutputCount,
	message := "Stopped controller writes"
).ToBe(expected := 2);
assertions.ThatInt(
	actual := _OutputStopController.AfterOutputCount,
	message := "Stopped controller finishes"
).ToBe(expected := 1);
END_METHOD

(*!
<summary>Checks sibling writes under Ignore and Continue and interruption after a stop/reset callback.</summary>
<param name="assertions">Valid assertion context borrowed from the active case.</param>
*)
METHOD PRIVATE testOutputPhaseContinuation
VAR_INPUT
	assertions : REFERENCE TO TOF_Testing.Assertions;
END_VAR
_OutputPoliciesBranch.Initialize();
_OutputPoliciesBranch.ChildCriticalErrorHandlingPolicy := TOF_Automation.ChildCriticalErrorHandlingPolicies.Ignore;
_OutputPoliciesBranch.ChildA.ThrowOnNextOutput := TRUE;
_OutputPoliciesBranch.ProcessOutput();
assertions.ThatInt(
	actual := _OutputPoliciesBranch.ChildB.ProcessOutputCount,
	message := "Ignore reaches next output"
).ToBe(expected := 1);
assertions.ThatInt(
	actual := _OutputPoliciesBranch.AfterOutputCount,
	message := "Ignore completes the pass"
).ToBe(expected := 1);

_OutputPoliciesBranch.ChildCriticalErrorHandlingPolicy :=
	TOF_Automation.ChildCriticalErrorHandlingPolicies.SetErrorAndContinue;
_OutputPoliciesBranch.ProcessOutput();
assertions.ThatInt(
	actual := _OutputPoliciesBranch.ChildB.ProcessOutputCount,
	message := "Continue reaches next output"
).ToBe(expected := 2);
assertions.ThatInt(
	actual := _OutputPoliciesBranch.AfterOutputCount,
	message := "Continue completes the pass"
).ToBe(expected := 2);

_OutputPoliciesBranch.StopAndResetBeforeOutput := TRUE;
_OutputPoliciesBranch.ProcessOutput();
assertions.ThatBool(
	actual := _OutputPoliciesBranch.OperationalState = TOF_Automation.OPERATIONAL_STATE.WORKING,
	message := "Reset restored work"
).IsTrue();
assertions.ThatInt(
	actual := _OutputPoliciesBranch.ChildA.ProcessOutputCount,
	message := "Obsolete pass skips first output"
).ToBe(expected := 2);
assertions.ThatInt(
	actual := _OutputPoliciesBranch.AfterOutputCount,
	message := "Obsolete pass skips after hook"
).ToBe(expected := 2);
END_METHOD

(*!
<summary>Checks the component snapshot after the real filter reuses the task-local native exception.</summary>
<param name="leaf">Fixture in the required lifecycle state.</param>
<param name="reaction">Runtime reaction under test.</param>
<param name="assertions">Valid assertion context borrowed from the active case.</param>
*)
METHOD PRIVATE checkPrimaryErrorCopy
VAR_INPUT
	assertions : REFERENCE TO TOF_Testing.Assertions;
	leaf : REFERENCE TO MockLeafAutomationComponent;
	reaction : TOF_Core.EXCEPTION_REACTION;
END_VAR
VAR
	primary : TOF_Core.IException;
	primaryMessage : TOF_Core.ERROR_MESSAGE;
	handlerThrew : BOOL;
END_VAR
primary := TOF_Core.ExceptionManager.GetLastException(
	exceptionCode := __SYSTEM.ExceptionCode.RTSEXCPT_ARRAYBOUNDS,
	catchPointNamespaceName := CurrentNamespace.Name,
	catchPointPOUName := __POUNAME(),
	catchPointPosition := __POSITION()
);
primaryMessage := primary.GetMessage();
MAIN.DiagnosticLogFilter.SetSecondaryExceptionProbe(enabled := TRUE);

__TRY
	leaf.ApplyExceptionReaction(exception := primary, reaction := reaction);
__CATCH
	handlerThrew := TRUE;
__ENDTRY

MAIN.DiagnosticLogFilter.SetSecondaryExceptionProbe(enabled := FALSE);
assertions.ThatBool(actual := handlerThrew, message := "Processing the native diagnostic must complete").IsFalse();
assertions.ThatBool(
	actual := primary.GetMessage() <> primaryMessage,
	message := "Filter must overwrite the borrowed wrapper"
).IsTrue();
assertions.ThatBool(
	actual := leaf.Error.TopMessage = primaryMessage,
	message := "Component must retain the primary message"
).IsTrue();
END_METHOD

(*!
<summary>Checks primary diagnostic capture for initialization, continue and stop reactions.</summary>
<description>Uses the installed test filter and task-local native wrapper without generating a hardware fault.</description>
<param name="assertions">Valid assertion context borrowed from the active case.</param>
*)
METHOD PRIVATE testPrimaryErrorBeforeLogging
VAR_INPUT
	assertions : REFERENCE TO TOF_Testing.Assertions;
END_VAR
checkPrimaryErrorCopy(
	assertions := assertions,
	leaf := _InitializingProbeLeaf,
	reaction := TOF_Core.EXCEPTION_REACTION.IGNORE
);
assertions.ThatBool(
	actual := _InitializingProbeLeaf.OperationalState = TOF_Automation.OPERATIONAL_STATE.INVALID
		AND_THEN _InitializingProbeLeaf.Error.Severity = TOF_Core.ERROR_SEVERITY.CRITICAL,
	message := "Initialization failure always records a critical error"
).IsTrue();

_WorkingProbeLeaf.Initialize();
checkPrimaryErrorCopy(
	assertions := assertions,
	leaf := _WorkingProbeLeaf,
	reaction := TOF_Core.EXCEPTION_REACTION.SET_ERROR_AND_CONTINUE
);
assertions.ThatBool(
	actual := _WorkingProbeLeaf.OperationalState = TOF_Automation.OPERATIONAL_STATE.WORKING
		AND_THEN _WorkingProbeLeaf.Error.Severity = TOF_Core.ERROR_SEVERITY.ERROR,
	message := "Continue records an error and keeps the component working"
).IsTrue();
checkPrimaryErrorCopy(
	assertions := assertions,
	leaf := _WorkingProbeLeaf,
	reaction := TOF_Core.EXCEPTION_REACTION.SET_ERROR_AND_STOP
);
assertions.ThatBool(
	actual := _WorkingProbeLeaf.OperationalState = TOF_Automation.OPERATIONAL_STATE.STOPPED
		AND_THEN _WorkingProbeLeaf.Error.Severity = TOF_Core.ERROR_SEVERITY.CRITICAL,
	message := "Stop replaces the lower severity error and stops the component"
).IsTrue();
END_METHOD

(*!
<summary>Checks input completion and stopped dispatch after the first input faults in a nested branch.</summary>
<param name="assertions">Valid assertion context borrowed from the active case.</param>
*)
METHOD PRIVATE testInputPhaseStop
VAR_INPUT
	assertions : REFERENCE TO TOF_Testing.Assertions;
END_VAR
_InputStopController.Children[0] := _InputStopBranch;
_InputStopController.ChildCriticalErrorHandlingPolicy :=
	TOF_Automation.ChildCriticalErrorHandlingPolicies.SetErrorAndStop;
_InputStopController.Initialize();
_InputStopBranch.ChildA.ThrowOnNextInput := TRUE;
_InputStopController.Execute();

assertions.ThatBool(
	actual := _InputStopController.OperationalState = TOF_Automation.OPERATIONAL_STATE.STOPPED
		AND_THEN _InputStopBranch.OperationalState = TOF_Automation.OPERATIONAL_STATE.STOPPED,
	message := "Critical input fault must stop both branches"
).IsTrue();
assertions.ThatInt(
	actual := _InputStopBranch.ChildB.ProcessInputCount,
	message := "Later input runs in the same scan"
).ToBe(expected := 1);
assertions.ThatInt(
	actual := _InputStopBranch.AfterInputCount,
	message := "Composite completes its input pass"
).ToBe(expected := 1);
assertions.ThatInt(
	actual := _InputStopController.AfterInputCount,
	message := "Controller completes its input pass"
).ToBe(expected := 1);
assertions.ThatInt(
	actual := _InputStopBranch.ChildB.WorkingCount,
	message := "Working logic must not follow the stop"
).ToBe(expected := 0);
END_METHOD

(*!
<summary>Checks that Reset and OnRecover failures always stop with a critical error regardless of policy.</summary>
<description>The branch fixture recovers from a copied error after explicitly resetting its stopped child.</description>
<param name="assertions">Valid assertion context borrowed from the active case.</param>
*)
METHOD PRIVATE testResetAndRecoverIgnoreExceptionPolicy
VAR_INPUT
	assertions : REFERENCE TO TOF_Testing.Assertions;
END_VAR
_ResetPolicyLeaf.Initialize();
_ResetPolicyLeaf.ExceptionHandlingPolicy := TOF_Core.ExceptionHandlingPolicies.SetErrorAndContinue;
_ResetPolicyLeaf.Stop(reason := "Policy test stop");
_ResetPolicyLeaf.ThrowOnReset := TRUE;
_ResetPolicyLeaf.Reset();
assertions.ThatDInt(
	actual := TO_DINT(_ResetPolicyLeaf.OperationalState),
	message := "Failed leaf OnReset must remain STOPPED even with SetErrorAndContinue"
).ToBe(expected := TO_DINT(TOF_Automation.OPERATIONAL_STATE.STOPPED));
assertions.ThatBool(
	actual := _ResetPolicyLeaf.HasError
		AND_THEN _ResetPolicyLeaf.Error.Severity = TOF_Core.ERROR_SEVERITY.CRITICAL,
	message := "Failed leaf OnReset must record a critical error"
).IsTrue();

_BeforeResetPolicyBranch.Initialize();
_BeforeResetPolicyBranch.ExceptionHandlingPolicy := TOF_Core.ExceptionHandlingPolicies.SetErrorAndContinue;
_BeforeResetPolicyBranch.Stop(reason := "Policy test stop");
_BeforeResetPolicyBranch.ThrowOnBeforeReset := TRUE;
_BeforeResetPolicyBranch.Reset();
assertions.ThatDInt(
	actual := TO_DINT(_BeforeResetPolicyBranch.OperationalState),
	message := "Failed OnBeforeChildrenReset must remain STOPPED even with SetErrorAndContinue"
).ToBe(expected := TO_DINT(TOF_Automation.OPERATIONAL_STATE.STOPPED));
assertions.ThatBool(
	actual := _BeforeResetPolicyBranch.HasError
		AND_THEN _BeforeResetPolicyBranch.Error.Severity = TOF_Core.ERROR_SEVERITY.CRITICAL,
	message := "Failed OnBeforeChildrenReset must record a critical error"
).IsTrue();
assertions.ThatInt(
	actual := _BeforeResetPolicyBranch.ChildA.ResetCount,
	message := "Failed OnBeforeChildrenReset must not reset children"
).ToBe(expected := 0);

_AfterResetPolicyBranch.Initialize();
_AfterResetPolicyBranch.ExceptionHandlingPolicy := TOF_Core.ExceptionHandlingPolicies.SetErrorAndContinue;
_AfterResetPolicyBranch.Stop(reason := "Policy test stop");
_AfterResetPolicyBranch.ThrowOnAfterReset := TRUE;
_AfterResetPolicyBranch.Reset();
assertions.ThatDInt(
	actual := TO_DINT(_AfterResetPolicyBranch.OperationalState),
	message := "Failed OnAfterChildrenReset must remain STOPPED even with SetErrorAndContinue"
).ToBe(expected := TO_DINT(TOF_Automation.OPERATIONAL_STATE.STOPPED));
assertions.ThatBool(
	actual := _AfterResetPolicyBranch.HasError
		AND_THEN _AfterResetPolicyBranch.Error.Severity = TOF_Core.ERROR_SEVERITY.CRITICAL,
	message := "Failed OnAfterChildrenReset must record a critical error"
).IsTrue();

_RecoverPolicyLeaf.Initialize();
_RecoverPolicyLeaf.ExceptionHandlingPolicy := TOF_Core.ExceptionHandlingPolicies.SetErrorAndContinue;
_RecoverPolicyLeaf.FailOnWorking := TRUE;
_RecoverPolicyLeaf.Execute();
_RecoverPolicyLeaf.FailOnWorking := FALSE;
_RecoverPolicyLeaf.ThrowOnRecover := TRUE;
_RecoverPolicyLeaf.Execute();
assertions.ThatDInt(
	actual := TO_DINT(_RecoverPolicyLeaf.OperationalState),
	message := "Failed leaf OnRecover must stop even with SetErrorAndContinue"
).ToBe(expected := TO_DINT(TOF_Automation.OPERATIONAL_STATE.STOPPED));
assertions.ThatBool(
	actual := _RecoverPolicyLeaf.HasError
		AND_THEN _RecoverPolicyLeaf.Error.Severity = TOF_Core.ERROR_SEVERITY.CRITICAL,
	message := "Failed leaf OnRecover must record a critical error"
).IsTrue();
assertions.ThatInt(
	actual := _RecoverPolicyLeaf.RecoverCount,
	message := "Leaf OnRecover must run once"
).ToBe(expected := 1);
assertions.ThatInt(
	actual := _RecoverPolicyLeaf.WorkingCount,
	message := "Failed leaf OnRecover must skip OnWorking"
).ToBe(expected := 1);

_RecoverPolicyBranch.Initialize();
_RecoverPolicyBranch.ExceptionHandlingPolicy := TOF_Core.ExceptionHandlingPolicies.SetErrorAndContinue;
_RecoverPolicyBranch.ChildCriticalErrorHandlingPolicy :=
	TOF_Automation.ChildCriticalErrorHandlingPolicies.SetErrorAndContinue;
_RecoverPolicyBranch.ChildA.ExceptionHandlingPolicy := TOF_Core.ExceptionHandlingPolicies.SetErrorAndStop;
_RecoverPolicyBranch.ChildA.FailOnWorking := TRUE;
_RecoverPolicyBranch.Execute();
assertions.ThatBool(
	actual := _RecoverPolicyBranch.ChildA.OperationalState = TOF_Automation.OPERATIONAL_STATE.STOPPED
		AND_THEN _RecoverPolicyBranch.ChildA.HasError
		AND_THEN _RecoverPolicyBranch.ChildA.Error.Severity = TOF_Core.ERROR_SEVERITY.CRITICAL,
	message := "The injected working failure must stop the child with a critical error"
).IsTrue();
assertions.ThatBool(
	actual := _RecoverPolicyBranch.OperationalState = TOF_Automation.OPERATIONAL_STATE.WORKING
		AND_THEN _RecoverPolicyBranch.HasError
		AND_THEN _RecoverPolicyBranch.Error.Severity = TOF_Core.ERROR_SEVERITY.ERROR,
	message := "The branch must stay working with a copied error until the child resets"
).IsTrue();

_RecoverPolicyBranch.ChildA.FailOnWorking := FALSE;
_RecoverPolicyBranch.ChildA.Reset();
_RecoverPolicyBranch.ThrowOnRecover := TRUE;
_RecoverPolicyBranch.Execute();
assertions.ThatDInt(
	actual := TO_DINT(_RecoverPolicyBranch.OperationalState),
	message := "Failed branch OnRecover must stop even with SetErrorAndContinue"
).ToBe(expected := TO_DINT(TOF_Automation.OPERATIONAL_STATE.STOPPED));
assertions.ThatBool(
	actual := _RecoverPolicyBranch.HasError
		AND_THEN _RecoverPolicyBranch.Error.Severity = TOF_Core.ERROR_SEVERITY.CRITICAL,
	message := "Failed branch OnRecover must record a critical error"
).IsTrue();
assertions.ThatInt(
	actual := _RecoverPolicyBranch.RecoverCount,
	message := "Branch OnRecover must run once"
).ToBe(expected := 1);
assertions.ThatInt(
	actual := _RecoverPolicyBranch.ChildA.WorkingCount,
	message := "Failed branch OnRecover must skip children working traversal"
).ToBe(expected := 1);
assertions.ThatInt(
	actual := _RecoverPolicyBranch.ChildB.WorkingCount,
	message := "Failed branch OnRecover must skip later children working traversal"
).ToBe(expected := 1);
END_METHOD

(*!
<summary>Checks sequential child-to-branch initialization completion and timeout normalization.</summary>
<param name="assertions">Valid assertion context borrowed from the active case.</param>
*)
METHOD PRIVATE testAfterChildrenInitializingAndTimeoutPropagation
VAR_INPUT
	assertions : REFERENCE TO TOF_Testing.Assertions;
END_VAR
_AfterInitBranch.ChildA.InitReturnValue := FALSE;
_AfterInitBranch.AfterInitReturnValue := FALSE;
_AfterInitBranch.ChildB.InitializationTimeout := T#15S;

assertions.ThatBool(
	actual := _AfterInitBranch.Initialize(),
	message := "Branch remains initializing while ChildA is pending"
).IsFalse();
assertions.ThatInt(
	actual := _AfterInitBranch.AfterInitializeCount,
	message := "OnAfterChildrenInitializing must not run before all children initialize"
).ToBe(expected := 0);
assertions.ThatBool(
	actual := _AfterInitBranch.InitializationTimeout = T#15S,
	message := "Branch initialization timeout must expand to match child timeout"
).IsTrue();

_AfterInitBranch.ChildA.InitReturnValue := TRUE;
assertions.ThatBool(
	actual := _AfterInitBranch.Initialize(),
	message := "Branch remains initializing while OnAfterChildrenInitializing returns FALSE"
).IsFalse();
assertions.ThatInt(
	actual := _AfterInitBranch.AfterInitializeCount,
	message := "OnAfterChildrenInitializing runs once all children are ready"
).ToBe(expected := 1);
assertions.ThatDInt(
	actual := TO_DINT(_AfterInitBranch.OperationalState),
	message := "Branch stays INITIALIZING when OnAfterChildrenInitializing returns FALSE"
).ToBe(expected := TO_DINT(TOF_Automation.OPERATIONAL_STATE.INITIALIZING));

_AfterInitBranch.AfterInitReturnValue := TRUE;
assertions.ThatBool(
	actual := _AfterInitBranch.Initialize(),
	message := "Branch completes initialization when OnAfterChildrenInitializing returns TRUE"
).IsTrue();
assertions.ThatInt(
	actual := _AfterInitBranch.AfterInitializeCount,
	message := "OnAfterChildrenInitializing runs again to finish initialization"
).ToBe(expected := 2);
assertions.ThatDInt(
	actual := TO_DINT(_AfterInitBranch.OperationalState),
	message := "Branch transitions to WORKING once OnAfterChildrenInitializing succeeds"
).ToBe(expected := TO_DINT(TOF_Automation.OPERATIONAL_STATE.WORKING));

_TimeoutNormLeaf.InitializationTimeout := T#10S;
_TimeoutNormLeaf.InitializationTimeout := T#0S;
assertions.ThatBool(
	actual := _TimeoutNormLeaf.InitializationTimeout = TOF_Automation.Parameters.InitializationTimeout,
	message := "Assigning T#0S must immediately resolve InitializationTimeout to global default"
).IsTrue();
END_METHOD

(*!
<summary>Checks disabled child stop/reset/enable semantics and single-shot HMI command consumption.</summary>
<param name="assertions">Valid assertion context borrowed from the active case.</param>
*)
METHOD PRIVATE testDisabledChildStopResetAndHmiCommandConsumption
VAR_INPUT
	assertions : REFERENCE TO TOF_Testing.Assertions;
END_VAR
VAR
	exceptionCode : __SYSTEM.ExceptionCode;
	exceptionEscaped : BOOL;
END_VAR
_DisabledChildBranch.Initialize();
_DisabledChildBranch.ChildA.Disable();
_DisabledChildBranch.Stop(reason := "Branch stop with disabled child");
assertions.ThatDInt(
	actual := TO_DINT(_DisabledChildBranch.OperationalState),
	message := "Branch enters STOPPED"
).ToBe(expected := TO_DINT(TOF_Automation.OPERATIONAL_STATE.STOPPED));
assertions.ThatDInt(
	actual := TO_DINT(_DisabledChildBranch.ChildB.OperationalState),
	message := "Enabled child enters STOPPED"
).ToBe(expected := TO_DINT(TOF_Automation.OPERATIONAL_STATE.STOPPED));
assertions.ThatDInt(
	actual := TO_DINT(_DisabledChildBranch.ChildA.OperationalState),
	message := "Disabled WORKING child must also transition to STOPPED"
).ToBe(expected := TO_DINT(TOF_Automation.OPERATIONAL_STATE.STOPPED));

_DisabledChildBranch.Reset();
assertions.ThatDInt(
	actual := TO_DINT(_DisabledChildBranch.OperationalState),
	message := "Branch resumes WORKING on Reset"
).ToBe(expected := TO_DINT(TOF_Automation.OPERATIONAL_STATE.WORKING));
assertions.ThatDInt(
	actual := TO_DINT(_DisabledChildBranch.ChildB.OperationalState),
	message := "Enabled child resumes WORKING on Reset"
).ToBe(expected := TO_DINT(TOF_Automation.OPERATIONAL_STATE.WORKING));
assertions.ThatDInt(
	actual := TO_DINT(_DisabledChildBranch.ChildA.OperationalState),
	message := "Disabled child remains STOPPED when branch resets"
).ToBe(expected := TO_DINT(TOF_Automation.OPERATIONAL_STATE.STOPPED));
assertions.ThatInt(
	actual := _DisabledChildBranch.ChildA.ResetCount,
	message := "Disabled child must not execute OnReset during branch Reset"
).ToBe(expected := 0);

_DisabledChildBranch.ChildA.Enable(includeChildren := TRUE);
assertions.ThatBool(actual := _DisabledChildBranch.ChildA.Enabled, message := "ChildA is enabled").IsTrue();
assertions.ThatDInt(
	actual := TO_DINT(_DisabledChildBranch.ChildA.OperationalState),
	message := "Enabling a stopped child must not auto-reset it"
).ToBe(expected := TO_DINT(TOF_Automation.OPERATIONAL_STATE.STOPPED));

_DisabledChildBranch.ChildA.Reset();
assertions.ThatDInt(
	actual := TO_DINT(_DisabledChildBranch.ChildA.OperationalState),
	message := "Explicit Reset restores the re-enabled child to WORKING"
).ToBe(expected := TO_DINT(TOF_Automation.OPERATIONAL_STATE.WORKING));
assertions.ThatInt(
	actual := _DisabledChildBranch.ChildA.ResetCount,
	message := "Explicit Reset invokes OnReset once"
).ToBe(expected := 1);

_CmdHmiController.ConfigurePlugins(plugins := _CmdHmiPlugins);
_CmdHmiController.Initialize();
_CmdHmiPlugin.AutomationComponentCommands.Disable := TRUE;
_CmdHmiController.Execute();
assertions.ThatBool(
	actual := _CmdHmiController.Enabled,
	message := "HMI Disable succeeds before fault injection"
).IsFalse();

_CmdHmiController.Child.ThrowOnEnable := TRUE;
_CmdHmiPlugin.AutomationComponentCommands.Enable := TRUE;

__TRY
	_CmdHmiController.Execute();
__CATCH(exceptionCode)
	exceptionEscaped := TRUE;
__ENDTRY

assertions.ThatBool(
	actual := exceptionEscaped,
	message := "Controller cycle service contains plugin Enable failure"
).IsFalse();
assertions.ThatBool(
	actual := _CmdHmiPlugin.AutomationComponentCommands.Enable,
	message := "HMI Enable flag must be cleared even when Enable raises an exception"
).IsFalse();
assertions.ThatBool(
	actual := _CmdHmiController.HasError,
	message := "Controller records the failed Enable command error"
).IsTrue();
assertions.ThatBool(
	actual := _CmdHmiController.Enabled,
	message := "Failed Enable must leave controller disabled"
).IsFalse();

_CmdHmiController.Execute();
assertions.ThatInt(
	actual := _CmdHmiController.Child.EnableCount,
	message := "Consumed HMI Enable command must not repeat on subsequent cycles"
).ToBe(expected := 1);
END_METHOD

(*!
<summary>Advances one cycle of the initialization timeout scenario.</summary>
<description>Reports the child error and INVALID state. Fifty calls bound lack of progress.</description>
<param name="assertions">Valid assertion context borrowed from the active case.</param>
*)
METHOD AdvanceInitializationTimeout : TOF_Testing.TEST_CYCLE_RESULT
VAR_INPUT
	assertions : REFERENCE TO TOF_Testing.Assertions;
END_VAR
VAR_INST
	cycleCount : INT;
END_VAR
AdvanceInitializationTimeout := TOF_Testing.TEST_CYCLE_RESULT.DONE;

IF cycleCount = 0 THEN
	_TimeoutComposite.ChildA.InitReturnValue := FALSE;
	_TimeoutComposite.ChildA.InitializationTimeout := T#1MS;
	_TimeoutComposite.InitializationTimeout := T#5S;
END_IF

cycleCount := cycleCount + 1;
_TimeoutComposite.Initialize();

IF _TimeoutComposite.ChildA.OperationalState = TOF_Automation.OPERATIONAL_STATE.INVALID OR_ELSE cycleCount >= 50 THEN
	assertions.ThatBool(
		actual := _TimeoutComposite.ChildA.HasError,
		message := TO_WSTRING(TOF_Core.Strings.Concat255(
			'Child timeout: child=', TO_STRING(_TimeoutComposite.ChildA.OperationalState),
			', parent=', TO_STRING(_TimeoutComposite.OperationalState),
			', PT=', TO_STRING(_TimeoutComposite.ChildA.InitializationTimeout),
			', init calls=', TO_STRING(_TimeoutComposite.ChildA.InitializeCount),
			', returns=', TO_STRING(_TimeoutComposite.ChildA.InitReturnValue)
		))
	).IsTrue();
	assertions.ThatDInt(
		actual := TO_DINT(_TimeoutComposite.ChildA.OperationalState),
		message := "Initialization timeout must put the child in INVALID"
	).ToBe(expected := TO_DINT(TOF_Automation.OPERATIONAL_STATE.INVALID));
	assertions.ThatBool(
		actual := _TimeoutComposite.ChildA.InitializeCount > 1,
		message := "The parent must allow repeated child initialization before timeout"
	).IsTrue();
ELSE
	AdvanceInitializationTimeout := TOF_Testing.TEST_CYCLE_RESULT.BUSY;
END_IF
END_METHOD

END_FUNCTION_BLOCK

// ---- Tests/Automation/MockCompositeAutomationComponent.TcPOU
(*
SPDX-FileCopyrightText: © 2026 Oleksandr Tiutyk <trofimich@gmail.com>
SPDX-License-Identifier: MIT
License: https://opensource.org/license/mit
*)

(*!
<summary>Mock composite with two leaves, callback observations and explicit storage faults.</summary>
<description>Self-bound child relationships require a live instance that is not copied.</description>
*)

FUNCTION_BLOCK MockCompositeAutomationComponent EXTENDS TOF_Automation.CompositeAutomationComponent<2>
VAR_OUTPUT
	//! <summary>Number of completed output passes observed by the after-output hook.</summary>
	AfterOutputCount : INT;
	//! <summary>Counts completed input passes.</summary>
	AfterInputCount : INT;
END_VAR
VAR_INPUT
	//! <summary>Stops and immediately resets this branch in the opening output hook.</summary>
	StopAndResetBeforeOutput : BOOL;
END_VAR
VAR_STAT
	{attribute 'hide'}
	_ClassName : STRING := __POUNAME();
END_VAR
VAR
	_ChildA : MockLeafAutomationComponent(name := "ChildA", parent := THIS^);
	_ChildB : MockLeafAutomationComponent(name := "ChildB", parent := THIS^);
	
	_Children : ARRAY [0.._ChildCount - 1] OF TOF_Automation.IChildAutomationComponent :=
	[
		_ChildA,
		_ChildB
	];
	
	_ThrowOnGetChildren : BOOL;
	_MissingChildrenReference : BOOL;
	_ResetOnBeforeChildrenStopped : BOOL;
	_BeforeInitializeCount : INT;
	_AfterWorkingCount : INT;

	_EventReceivedCount : INT;
	_LastReceivedEventId : INT;
	_AfterInitializeCount : INT;
	_AfterInitReturnValue : BOOL := TRUE;
	_RecoverCount : INT;
	_ThrowOnRecover : BOOL;
	_ThrowOnBeforeReset : BOOL;
	_ThrowOnAfterReset : BOOL;
END_VAR

{attribute 'monitoring' := 'call'}
PROPERTY ChildA : REFERENCE TO MockLeafAutomationComponent
GET
ChildA REF= _ChildA;
END_GET
END_PROPERTY

{attribute 'monitoring' := 'call'}
PROPERTY ChildB : REFERENCE TO MockLeafAutomationComponent
GET
ChildB REF= _ChildB;
END_GET
END_PROPERTY

(*!
<summary>Returns test child storage or the configured missing/throwing fault.</summary>
<description>
The borrowed array and its self-bound children must not be copied. Faults exercise lookup containment
and validation before initialization hooks.
</description>
*)
{attribute 'monitoring' := 'call'}
PROPERTY FINAL Children : REFERENCE TO ARRAY [0.._ChildCount - 1] OF TOF_Automation.IChildAutomationComponent
GET
IF _ThrowOnGetChildren THEN
	TOF_Core.Exceptions.ThrowStandard(
		sourceNamespaceName := NamespaceName,
		sourceClassName := ClassName,
		sourcePOUName := __POUNAME(),
		sourcePosition := __POSITION(),
		message := "Injected Children getter failure."
	);
END_IF

IF _MissingChildrenReference THEN
	Children REF= 0;
ELSE
	Children REF= _Children;
END_IF
END_GET
END_PROPERTY

{attribute 'monitoring' := 'call'}
PROPERTY ClassName : REFERENCE TO STRING
GET
ClassName REF= _ClassName;
END_GET
END_PROPERTY

{attribute 'monitoring' := 'call'}
PROPERTY EventReceivedCount : INT
GET
EventReceivedCount := _EventReceivedCount;
END_GET
END_PROPERTY

METHOD FB_init : BOOL
VAR_INPUT
	bInitRetains : BOOL; // TRUE: the retain variables are initialized (reset warm / reset cold)
	bInCopyCode : BOOL;  // TRUE: the instance will be copied to the copy code afterward (online change)
	name : WSTRING;
	parent : TOF_Automation.IParentAutomationComponent;
END_VAR
END_METHOD

{attribute 'monitoring' := 'call'}
PROPERTY LastReceivedEventId : INT
GET
LastReceivedEventId := _LastReceivedEventId;
END_GET
END_PROPERTY

{attribute 'monitoring' := 'call'}
PROPERTY NamespaceName : REFERENCE TO STRING
GET
NamespaceName REF= CurrentNamespace.Name;
END_GET
END_PROPERTY

METHOD OnEventReceived
VAR_INPUT
	event : TOF_Core.IEvent;
END_VAR
VAR_OUTPUT
	stopPropagation : BOOL;
END_VAR
VAR
	mockEv : POINTER TO MockAutomationEvent;
END_VAR
_EventReceivedCount := _EventReceivedCount + 1;

IF __QUERYPOINTER(event, mockEv) THEN
	_LastReceivedEventId := mockEv^.EventId;
END_IF

stopPropagation := FALSE;
END_METHOD

{attribute 'monitoring' := 'call'}
PROPERTY SelfSize : ULINT
GET
SelfSize := XSIZEOF(THIS^);
END_GET
END_PROPERTY

(*!
<summary>Controls an exception from the Children getter.</summary>
*)
{attribute 'monitoring' := 'call'}
PROPERTY ThrowOnGetChildren : BOOL
GET
ThrowOnGetChildren := _ThrowOnGetChildren;
END_GET
SET
_ThrowOnGetChildren := ThrowOnGetChildren;
END_SET
END_PROPERTY

(*!
<summary>Controls a missing Children storage reference.</summary>
*)
{attribute 'monitoring' := 'call'}
PROPERTY MissingChildrenReference : BOOL
GET
MissingChildrenReference := _MissingChildrenReference;
END_GET
SET
_MissingChildrenReference := MissingChildrenReference;
END_SET
END_PROPERTY

(*!
<summary>Requests one Reset from the next before-stopped hook.</summary>
*)
{attribute 'monitoring' := 'call'}
PROPERTY ResetOnBeforeChildrenStopped : BOOL
GET
ResetOnBeforeChildrenStopped := _ResetOnBeforeChildrenStopped;
END_GET
SET
_ResetOnBeforeChildrenStopped := ResetOnBeforeChildrenStopped;
END_SET
END_PROPERTY

(*!
<summary>Gets the number of completed BeforeInitialize hook calls.</summary>
*)
PROPERTY BeforeInitializeCount : INT
GET
BeforeInitializeCount := _BeforeInitializeCount;
END_GET
END_PROPERTY

(*!
<summary>Gets the number of completed AfterWorking hook calls.</summary>
*)
PROPERTY AfterWorkingCount : INT
GET
AfterWorkingCount := _AfterWorkingCount;
END_GET
END_PROPERTY

(*!
<summary>Records entry into the branch initialization hook.</summary>
*)
METHOD PROTECTED OnBeforeChildrenInitializing
_BeforeInitializeCount := _BeforeInitializeCount + 1;
END_METHOD

(*!
<summary>Records completion of working-child traversal.</summary>
*)
METHOD PROTECTED OnAfterChildrenWorking
_AfterWorkingCount := _AfterWorkingCount + 1;
END_METHOD

(*!
<summary>Optionally resumes the tree from within its stopped-cycle callback.</summary>
<description>
Consumes the request before Reset so it cannot trigger a repeated request from this hook.
</description>
*)
METHOD PROTECTED OnBeforeChildrenStopped
IF _ResetOnBeforeChildrenStopped THEN
	_ResetOnBeforeChildrenStopped := FALSE;
	Reset();
END_IF
END_METHOD

(*!
<summary>Counts completed output passes.</summary>
*)
METHOD PROTECTED OnAfterChildrenProcessOutput
AfterOutputCount := AfterOutputCount + 1;
END_METHOD

(*!
<summary>Optionally changes state twice before the first output.</summary>
*)
METHOD PROTECTED OnBeforeChildrenProcessOutput
IF StopAndResetBeforeOutput THEN
	Stop(reason := "Injected stop before output");
	Reset();
END_IF
END_METHOD

(*! <summary>Records completion of this branch's input traversal.</summary> *)
METHOD PROTECTED OnAfterChildrenProcessInput
AfterInputCount := AfterInputCount + 1;
END_METHOD

(*!
<summary>Counts after-children initialization calls and returns the configured completion flag.</summary>
*)
METHOD PROTECTED OnAfterChildrenInitializing : BOOL
_AfterInitializeCount := _AfterInitializeCount + 1;
OnAfterChildrenInitializing := _AfterInitReturnValue;
END_METHOD

(*!
<summary>Optionally raises a fault during the after-children reset hook.</summary>
*)
METHOD PROTECTED OnAfterChildrenReset
IF _ThrowOnAfterReset THEN
	TOF_Core.Exceptions.ThrowStandard(
		sourceNamespaceName := NamespaceName,
		sourceClassName := ClassName,
		sourcePOUName := __POUNAME(),
		sourcePosition := __POSITION(),
		message := "Injected OnAfterChildrenReset failure."
	);
END_IF
END_METHOD

(*!
<summary>Optionally raises a fault during the before-children reset hook.</summary>
*)
METHOD PROTECTED OnBeforeChildrenReset
IF _ThrowOnBeforeReset THEN
	TOF_Core.Exceptions.ThrowStandard(
		sourceNamespaceName := NamespaceName,
		sourceClassName := ClassName,
		sourcePOUName := __POUNAME(),
		sourcePosition := __POSITION(),
		message := "Injected OnBeforeChildrenReset failure."
	);
END_IF
END_METHOD

(*!
<summary>Records OnRecover calls and optionally raises a recovery fault.</summary>
*)
METHOD PROTECTED OnRecover
_RecoverCount := _RecoverCount + 1;

IF _ThrowOnRecover THEN
	TOF_Core.Exceptions.ThrowStandard(
		sourceNamespaceName := NamespaceName,
		sourceClassName := ClassName,
		sourcePOUName := __POUNAME(),
		sourcePosition := __POSITION(),
		message := "Injected branch OnRecover failure."
	);
END_IF
END_METHOD

(*!
<summary>Gets the number of completed OnAfterChildrenInitializing hook calls.</summary>
*)
{attribute 'monitoring' := 'call'}
PROPERTY AfterInitializeCount : INT
GET
AfterInitializeCount := _AfterInitializeCount;
END_GET
END_PROPERTY

(*!
<summary>Controls the return value of OnAfterChildrenInitializing.</summary>
*)
{attribute 'monitoring' := 'call'}
PROPERTY AfterInitReturnValue : BOOL
GET
AfterInitReturnValue := _AfterInitReturnValue;
END_GET
SET
_AfterInitReturnValue := AfterInitReturnValue;
END_SET
END_PROPERTY

(*!
<summary>Gets the number of OnRecover calls recorded by this mock composite.</summary>
*)
{attribute 'monitoring' := 'call'}
PROPERTY RecoverCount : INT
GET
RecoverCount := _RecoverCount;
END_GET
END_PROPERTY

(*!
<summary>Controls the OnAfterChildrenReset fault injected by regression tests.</summary>
*)
{attribute 'monitoring' := 'call'}
PROPERTY ThrowOnAfterReset : BOOL
GET
ThrowOnAfterReset := _ThrowOnAfterReset;
END_GET
SET
_ThrowOnAfterReset := ThrowOnAfterReset;
END_SET
END_PROPERTY

(*!
<summary>Controls the OnBeforeChildrenReset fault injected by regression tests.</summary>
*)
{attribute 'monitoring' := 'call'}
PROPERTY ThrowOnBeforeReset : BOOL
GET
ThrowOnBeforeReset := _ThrowOnBeforeReset;
END_GET
SET
_ThrowOnBeforeReset := ThrowOnBeforeReset;
END_SET
END_PROPERTY

(*!
<summary>Controls the OnRecover fault injected by regression tests.</summary>
*)
{attribute 'monitoring' := 'call'}
PROPERTY ThrowOnRecover : BOOL
GET
ThrowOnRecover := _ThrowOnRecover;
END_GET
SET
_ThrowOnRecover := ThrowOnRecover;
END_SET
END_PROPERTY

END_FUNCTION_BLOCK

// ---- Tests/Automation/MockLeafAutomationComponent.TcPOU
(*
SPDX-FileCopyrightText: © 2026 Oleksandr Tiutyk <trofimich@gmail.com>
SPDX-License-Identifier: MIT
License: https://opensource.org/license/mit
*)

(*!
<summary>Mock leaf for lifecycle hooks, I/O phases, initialization/reset faults and event routing.</summary>
*)

FUNCTION_BLOCK MockLeafAutomationComponent EXTENDS TOF_Automation.InputOutputLeafAutomationComponent
VAR_INPUT
	//! <summary>Raises one output fault after the output call has been counted.</summary>
	ThrowOnNextOutput : BOOL;
	//! <summary>Raises one fault during input acquisition.</summary>
	ThrowOnNextInput : BOOL;
END_VAR
VAR_STAT
	{attribute 'hide'}
	_ClassName : STRING := __POUNAME();
END_VAR
VAR
	{attribute 'hide'}
	_InitializeCount : INT;
	{attribute 'hide'}
	_WorkingCount : INT;
	{attribute 'hide'}
	_ProcessInputCount : INT;
	{attribute 'hide'}
	_ProcessOutputCount : INT;
	{attribute 'hide'}
	_ResetCount : INT;
	{attribute 'hide'}
	_StopCount : INT;
	{attribute 'hide'}
	_EnableCount : INT;
	{attribute 'hide'}
	_DisableCount : INT;
	{attribute 'hide'}
	_EventReceivedCount : INT;
	{attribute 'hide'}
	_LastReceivedEventId : INT;
	{attribute 'hide'}
	_StopPropagationOnEvent : BOOL;
	{attribute 'hide'}
	_InitReturnValue : BOOL := TRUE;
	{attribute 'hide'}
	_FailOnWorking : BOOL;
	_ThrowOnInitializing : BOOL;
	_ThrowOnReset : BOOL;
	_RecoverCount : INT;
	_ThrowOnRecover : BOOL;
	_ThrowOnEnable : BOOL;
	_ThrowOnDisable : BOOL;
END_VAR

{attribute 'monitoring' := 'call'}
PROPERTY ClassName : REFERENCE TO STRING
GET
ClassName REF= _ClassName;
END_GET
END_PROPERTY

{attribute 'monitoring' := 'call'}
PROPERTY DisableCount : INT
GET
DisableCount := _DisableCount;
END_GET
END_PROPERTY

{attribute 'monitoring' := 'call'}
PROPERTY EnableCount : INT
GET
EnableCount := _EnableCount;
END_GET
END_PROPERTY

{attribute 'monitoring' := 'call'}
PROPERTY EventReceivedCount : INT
GET
EventReceivedCount := _EventReceivedCount;
END_GET
END_PROPERTY

{attribute 'monitoring' := 'call'}
PROPERTY FailOnWorking : BOOL
GET
FailOnWorking := _FailOnWorking;
END_GET
SET
_FailOnWorking := FailOnWorking;
END_SET
END_PROPERTY

METHOD FB_init : BOOL
VAR_INPUT
	bInitRetains : BOOL; // TRUE: the retain variables are initialized (reset warm / reset cold)
	bInCopyCode : BOOL;  // TRUE: the instance will be copied to the copy code afterward (online change)
	name : WSTRING;
	parent : TOF_Automation.IParentAutomationComponent;
END_VAR
END_METHOD

{attribute 'monitoring' := 'call'}
PROPERTY InitializeCount : INT
GET
InitializeCount := _InitializeCount;
END_GET
END_PROPERTY

{attribute 'monitoring' := 'call'}
PROPERTY InitReturnValue : BOOL
GET
InitReturnValue := _InitReturnValue;
END_GET
SET
_InitReturnValue := InitReturnValue;
END_SET
END_PROPERTY

{attribute 'monitoring' := 'call'}
PROPERTY LastReceivedEventId : INT
GET
LastReceivedEventId := _LastReceivedEventId;
END_GET
END_PROPERTY

{attribute 'monitoring' := 'call'}
PROPERTY NamespaceName : REFERENCE TO STRING
GET
NamespaceName REF= CurrentNamespace.Name;
END_GET
END_PROPERTY

(*!
<summary>Records the OnDisable call and optionally injects an exception.</summary>
*)
METHOD PROTECTED OnDisable
_DisableCount := _DisableCount + 1;

IF _ThrowOnDisable THEN
	TOF_Core.Exceptions.ThrowStandard(
		sourceNamespaceName := NamespaceName,
		sourceClassName := ClassName,
		sourcePOUName := __POUNAME(),
		sourcePosition := __POSITION(),
		message := "Injected OnDisable failure."
	);
END_IF
END_METHOD

(*!
<summary>Records the OnEnable call and optionally injects an exception.</summary>
*)
METHOD PROTECTED OnEnable
_EnableCount := _EnableCount + 1;

IF _ThrowOnEnable THEN
	TOF_Core.Exceptions.ThrowStandard(
		sourceNamespaceName := NamespaceName,
		sourceClassName := ClassName,
		sourcePOUName := __POUNAME(),
		sourcePosition := __POSITION(),
		message := "Injected OnEnable failure."
	);
END_IF
END_METHOD

METHOD OnEventReceived
VAR_INPUT
	event : TOF_Core.IEvent;
END_VAR
VAR_OUTPUT
	stopPropagation : BOOL;
END_VAR
VAR
	mockEv : POINTER TO MockAutomationEvent;
END_VAR
_EventReceivedCount := _EventReceivedCount + 1;

IF __QUERYPOINTER(event, mockEv) THEN
	_LastReceivedEventId := mockEv^.EventId;
END_IF

stopPropagation := _StopPropagationOnEvent;
END_METHOD

(*!
<summary>Records the OnInitializing call and optionally injects an exception.</summary>
<description>
The exception exercises production conversion into a copied component error; the hook does not own it.
</description>
*)
METHOD PROTECTED OnInitializing : BOOL
_InitializeCount := _InitializeCount + 1;

IF _ThrowOnInitializing THEN
	TOF_Core.Exceptions.ThrowStandard(
		sourceNamespaceName := NamespaceName,
		sourceClassName := ClassName,
		sourcePOUName := __POUNAME(),
		sourcePosition := __POSITION(),
		message := "Injected OnInitializing failure."
	);
END_IF

OnInitializing := _InitReturnValue;
END_METHOD

(*! <summary>Counts input calls and raises an armed input fault once.</summary> *)
METHOD PROTECTED OnProcessInput
_ProcessInputCount := _ProcessInputCount + 1;

IF ThrowOnNextInput THEN
	ThrowOnNextInput := FALSE;
	TOF_Core.Exceptions.ThrowStandard(
		sourceNamespaceName := NamespaceName,
		sourceClassName := ClassName,
		sourcePOUName := __POUNAME(),
		sourcePosition := __POSITION(),
		message := "Injected input failure"
	);
END_IF
END_METHOD

(*! <summary>Counts output calls and optionally injects a one-shot fault after the observed effect.</summary> *)
METHOD PROTECTED OnProcessOutput
_ProcessOutputCount := _ProcessOutputCount + 1;

IF ThrowOnNextOutput THEN
	ThrowOnNextOutput := FALSE;
	TOF_Core.Exceptions.ThrowStandard(
		sourceNamespaceName := NamespaceName,
		sourceClassName := ClassName,
		sourcePOUName := __POUNAME(),
		sourcePosition := __POSITION(),
		message := "Injected output failure"
	);
END_IF
END_METHOD

(*!
<summary>Records the OnRecover call and optionally injects an exception.</summary>
*)
METHOD PROTECTED OnRecover
_RecoverCount := _RecoverCount + 1;

IF _ThrowOnRecover THEN
	TOF_Core.Exceptions.ThrowStandard(
		sourceNamespaceName := NamespaceName,
		sourceClassName := ClassName,
		sourcePOUName := __POUNAME(),
		sourcePosition := __POSITION(),
		message := "Injected OnRecover failure."
	);
END_IF
END_METHOD

(*!
<summary>Records the OnReset call and optionally injects an exception.</summary>
<description>
The exception exercises production conversion into a copied component error; the hook does not own it.
</description>
*)
METHOD PROTECTED OnReset
_ResetCount := _ResetCount + 1;

IF _ThrowOnReset THEN
	TOF_Core.Exceptions.ThrowStandard(
		sourceNamespaceName := NamespaceName,
		sourceClassName := ClassName,
		sourcePOUName := __POUNAME(),
		sourcePosition := __POSITION(),
		message := "Injected OnReset failure."
	);
END_IF
END_METHOD

METHOD PROTECTED OnStopped
_StopCount := _StopCount + 1;
END_METHOD

METHOD PROTECTED OnWorking
_WorkingCount := _WorkingCount + 1;

IF _FailOnWorking THEN
	TOF_Core.Exceptions.ThrowStandard(
		sourceNamespaceName := NamespaceName,
		sourceClassName := ClassName,
		sourcePOUName := __POUNAME(),
		sourcePosition := __POSITION(),
		message := "Mock leaf failure on working"
	);
END_IF
END_METHOD

{attribute 'monitoring' := 'call'}
PROPERTY ProcessInputCount : INT
GET
ProcessInputCount := _ProcessInputCount;
END_GET
END_PROPERTY

{attribute 'monitoring' := 'call'}
PROPERTY ProcessOutputCount : INT
GET
ProcessOutputCount := _ProcessOutputCount;
END_GET
END_PROPERTY

{attribute 'monitoring' := 'call'}
PROPERTY ResetCount : INT
GET
ResetCount := _ResetCount;
END_GET
END_PROPERTY

{attribute 'monitoring' := 'call'}
PROPERTY SelfSize : ULINT
GET
SelfSize := XSIZEOF(THIS^);
END_GET
END_PROPERTY

{attribute 'monitoring' := 'call'}
PROPERTY StopCount : INT
GET
StopCount := _StopCount;
END_GET
END_PROPERTY

{attribute 'monitoring' := 'call'}
PROPERTY StopPropagationOnEvent : BOOL
GET
StopPropagationOnEvent := _StopPropagationOnEvent;
END_GET
SET
_StopPropagationOnEvent := StopPropagationOnEvent;
END_SET
END_PROPERTY

{attribute 'monitoring' := 'call'}
PROPERTY WorkingCount : INT
GET
WorkingCount := _WorkingCount;
END_GET
END_PROPERTY

(*!
<summary>Controls the initialization-hook failure injected by regression tests.</summary>
*)
{attribute 'monitoring' := 'call'}
PROPERTY ThrowOnInitializing : BOOL
GET
ThrowOnInitializing := _ThrowOnInitializing;
END_GET
SET
_ThrowOnInitializing := ThrowOnInitializing;
END_SET
END_PROPERTY

(*!
<summary>Controls the reset-hook failure injected by regression tests.</summary>
*)
{attribute 'monitoring' := 'call'}
PROPERTY ThrowOnReset : BOOL
GET
ThrowOnReset := _ThrowOnReset;
END_GET
SET
_ThrowOnReset := ThrowOnReset;
END_SET
END_PROPERTY

(*!
<summary>Gets the number of OnRecover calls recorded by this mock leaf.</summary>
*)
{attribute 'monitoring' := 'call'}
PROPERTY RecoverCount : INT
GET
RecoverCount := _RecoverCount;
END_GET
END_PROPERTY

(*!
<summary>Controls the disable-hook failure injected by regression tests.</summary>
*)
{attribute 'monitoring' := 'call'}
PROPERTY ThrowOnDisable : BOOL
GET
ThrowOnDisable := _ThrowOnDisable;
END_GET
SET
_ThrowOnDisable := ThrowOnDisable;
END_SET
END_PROPERTY

(*!
<summary>Controls the enable-hook failure injected by regression tests.</summary>
*)
{attribute 'monitoring' := 'call'}
PROPERTY ThrowOnEnable : BOOL
GET
ThrowOnEnable := _ThrowOnEnable;
END_GET
SET
_ThrowOnEnable := ThrowOnEnable;
END_SET
END_PROPERTY

(*!
<summary>Controls the recover-hook failure injected by regression tests.</summary>
*)
{attribute 'monitoring' := 'call'}
PROPERTY ThrowOnRecover : BOOL
GET
ThrowOnRecover := _ThrowOnRecover;
END_GET
SET
_ThrowOnRecover := ThrowOnRecover;
END_SET
END_PROPERTY

(*!
<summary>Exercises the inherited exception handler with a borrowed diagnostic in the fixture's current state.</summary>
<param name="exception">Task-local exception that remains live for the call.</param>
<param name="reaction">Runtime reaction to apply.</param>
*)
METHOD ApplyExceptionReaction
VAR_INPUT
	exception : TOF_Core.IException;
	reaction : TOF_Core.EXCEPTION_REACTION;
END_VAR
ProcessException(exception := exception, exceptionReaction := reaction, exceptionSourceHint := "Injected primary failure");
END_METHOD

END_FUNCTION_BLOCK

// ---- Tests/Automation/MockAutomationEvent.TcPOU
(*
SPDX-FileCopyrightText: Â© 2026 Oleksandr Tiutyk <trofimich@gmail.com>
SPDX-License-Identifier: MIT
License: https://opensource.org/license/mit
*)

(*!
<summary>Mock event used for verifying event delivery and propagation in automation tests.</summary>
*)

FUNCTION_BLOCK MockAutomationEvent EXTENDS TOF_Core.Event
VAR_STAT
	{attribute 'hide'}
	_ClassName : STRING := __POUNAME();
END_VAR
VAR
	{attribute 'hide'}
	_EventId : INT;
	{attribute 'hide'}
	_Payload : WSTRING(255);
END_VAR

{attribute 'monitoring' := 'call'}
PROPERTY ClassName : REFERENCE TO STRING
GET
ClassName REF= _ClassName;
END_GET
END_PROPERTY

{attribute 'monitoring' := 'call'}
PROPERTY EventId : INT
GET
EventId := _EventId;
END_GET
END_PROPERTY

METHOD FB_init : BOOL
VAR_INPUT
	bInitRetains : BOOL; // TRUE: the retain variables are initialized (reset warm / reset cold)
	bInCopyCode : BOOL;  // TRUE: the instance will be copied to the copy code afterward (online change)
	sourceObject : TOF_Core.IObject;
	eventId : INT;
	payload : WSTRING(255);
END_VAR
_EventId := eventId;
_Payload := payload;
END_METHOD

{attribute 'monitoring' := 'call'}
PROPERTY NamespaceName : REFERENCE TO STRING
GET
NamespaceName REF= CurrentNamespace.Name;
END_GET
END_PROPERTY

{attribute 'monitoring' := 'call'}
PROPERTY Payload : REFERENCE TO WSTRING(255)
GET
Payload REF= _Payload;
END_GET
END_PROPERTY

{attribute 'monitoring' := 'call'}
PROPERTY SelfSize : ULINT
GET
SelfSize := XSIZEOF(THIS^);
END_GET
END_PROPERTY

END_FUNCTION_BLOCK

// ---- Tests/Automation/MockPluginAutomationController.TcPOU
(*
SPDX-FileCopyrightText: © 2026 Oleksandr Tiutyk <trofimich@gmail.com>
SPDX-License-Identifier: MIT
License: https://opensource.org/license/mit
*)

(*!
<summary>Hosts one leaf and borrowed plugins for controller-cycle regression tests.</summary>
<description>
Instances contain self-bound child interfaces and must not be copied. One task owns each instance;
plugin arrays must remain live for all calls that service them.
</description>
*)

{attribute 'no_explicit_call' := 'do not call this function block directly'}
FUNCTION_BLOCK MockPluginAutomationController EXTENDS TOF_Automation.AutomationController<1>
VAR_OUTPUT
	//! <summary>Number of completed output passes observed by the after-output hook.</summary>
	AfterOutputCount : INT;
	//! <summary>Counts completed input passes.</summary>
	AfterInputCount : INT;
END_VAR
VAR_STAT
	_ClassName : STRING := __POUNAME();
END_VAR
VAR
	_Child : MockLeafAutomationComponent(name := "PluginChild", parent := THIS^);
	_Children : ARRAY [0.._ChildCount - 1] OF TOF_Automation.IChildAutomationComponent := [_Child];
	_MissingChildrenReference : BOOL;
	_ThrowOnGetChildren : BOOL;
END_VAR

(*!
<summary>Borrows the static concrete class name.</summary>
*)
PROPERTY ClassName : REFERENCE TO STRING
GET
ClassName REF= _ClassName;
END_GET
END_PROPERTY

(*!
<summary>Borrows the library namespace.</summary>
*)
PROPERTY NamespaceName : REFERENCE TO STRING
GET
NamespaceName REF= CurrentNamespace.Name;
END_GET
END_PROPERTY

(*!
<summary>Gets the size of this complete root instance.</summary>
*)
PROPERTY SelfSize : ULINT
GET
SelfSize := XSIZEOF(THIS^);
END_GET
END_PROPERTY

(*!
<summary>Borrows the root-owned leaf for lifecycle and I/O observations.</summary>
*)
PROPERTY Child : REFERENCE TO MockLeafAutomationComponent
GET
Child REF= _Child;
END_GET
END_PROPERTY

(*!
<summary>Controls a missing child storage reference.</summary>
*)
{attribute 'monitoring' := 'call'}
PROPERTY MissingChildrenReference : BOOL
GET
MissingChildrenReference := _MissingChildrenReference;
END_GET
SET
_MissingChildrenReference := MissingChildrenReference;
END_SET
END_PROPERTY

(*!
<summary>Controls an exception from the Children getter.</summary>
*)
{attribute 'monitoring' := 'call'}
PROPERTY ThrowOnGetChildren : BOOL
GET
ThrowOnGetChildren := _ThrowOnGetChildren;
END_GET
SET
_ThrowOnGetChildren := ThrowOnGetChildren;
END_SET
END_PROPERTY

(*!
<summary>Borrows the root-owned child array or injects a configured getter fault.</summary>
*)
PROPERTY Children : REFERENCE TO ARRAY [0.._ChildCount - 1] OF TOF_Automation.IChildAutomationComponent
GET
IF _ThrowOnGetChildren THEN
	TOF_Core.Exceptions.ThrowStandard(
		sourceNamespaceName := NamespaceName,
		sourceClassName := ClassName,
		sourcePOUName := __POUNAME(),
		sourcePosition := __POSITION(),
		message := "Injected controller Children getter failure."
	);
END_IF

IF _MissingChildrenReference THEN
	Children REF= 0;
ELSE
	Children REF= _Children;
END_IF
END_GET
END_PROPERTY

(*!
<summary>Borrows a plugin array for the regression scenario.</summary>
<description>
The caller keeps the array and plugins live until this controller is no longer serviced. No ownership
is transferred. Call before execution from the owning task.
</description>
*)
METHOD ConfigurePlugins
VAR_IN_OUT CONSTANT
	plugins : ARRAY [*] OF TOF_Automation.IAutomationControllerPlugin;
END_VAR
AssignPlugins(plugins := plugins);
END_METHOD

(*!
<summary>Counts completed output passes.</summary>
*)
METHOD PROTECTED OnAfterChildrenProcessOutput
AfterOutputCount := AfterOutputCount + 1;
END_METHOD

(*! <summary>Records completion of this branch's input traversal.</summary> *)
METHOD PROTECTED OnAfterChildrenProcessInput
AfterInputCount := AfterInputCount + 1;
END_METHOD

END_FUNCTION_BLOCK

// ---- Tests/Automation/MockHmiControllerPlugin.TcPOU
(*
SPDX-FileCopyrightText: © 2026 Oleksandr Tiutyk <trofimich@gmail.com>
SPDX-License-Identifier: MIT
License: https://opensource.org/license/mit
*)

(*!
<summary>Dispatches HMI base commands and records both controller-service callbacks.</summary>
<description>
Uses the base HMI command and status storage. One task owns each instance; no controller reference
is retained between calls. An optional before-service fault exercises the controller exception policy.
</description>
*)

{attribute 'no_explicit_call' := 'do not call this function block directly'}
FUNCTION_BLOCK MockHmiControllerPlugin EXTENDS TOF_Automation.HmiAutomationComponentElement
	IMPLEMENTS TOF_Automation.IAutomationControllerPlugin
VAR_STAT
	_ClassName : STRING := __POUNAME();
END_VAR
VAR
	_BeforeCount : INT;
	_AfterCount : INT;
	_ThrowOnBeforeExecute : BOOL;
END_VAR

(*!
<summary>Borrows the static concrete class name.</summary>
*)
PROPERTY ClassName : REFERENCE TO STRING
GET
ClassName REF= _ClassName;
END_GET
END_PROPERTY

(*!
<summary>Borrows the library namespace.</summary>
*)
PROPERTY NamespaceName : REFERENCE TO STRING
GET
NamespaceName REF= CurrentNamespace.Name;
END_GET
END_PROPERTY

(*!
<summary>Gets the number of completed Before hook calls.</summary>
*)
PROPERTY BeforeCount : INT
GET
BeforeCount := _BeforeCount;
END_GET
END_PROPERTY

(*!
<summary>Gets the number of completed After hook calls.</summary>
*)
PROPERTY AfterCount : INT
GET
AfterCount := _AfterCount;
END_GET
END_PROPERTY

(*!
<summary>Records the before callback, optionally fails, and dispatches HMI commands.</summary>
<description>
The injected exception exercises stop policy while disabled. This callback never performs technological
work and retains no exception or controller reference.
</description>
*)
METHOD OnBeforeControllerExecute
VAR_INPUT
	controller : TOF_Automation.IAutomationController;
END_VAR
_BeforeCount := _BeforeCount + 1;
IF _ThrowOnBeforeExecute THEN
	TOF_Core.Exceptions.ThrowStandard(
		sourceNamespaceName := NamespaceName,
		sourceClassName := ClassName,
		sourcePOUName := __POUNAME(),
		sourcePosition := __POSITION(),
		message := "Injected before-plugin service failure."
	);
END_IF

ProcessAutomationComponentCommands(automationComponent := controller);
END_METHOD

(*!
<summary>Records the after callback and services HMI statuses.</summary>
<description>
Runs even while disabled; this callback performs service only and does not execute technological work.
</description>
*)
METHOD OnAfterControllerExecute
VAR_INPUT
	controller : TOF_Automation.IAutomationController;
END_VAR
_AfterCount := _AfterCount + 1;
UpdateAutomationComponentStatuses(automationComponent := controller);
END_METHOD

(*!
<summary>Controls a failure before HMI command dispatch.</summary>
*)
PROPERTY ThrowOnBeforeExecute : BOOL
GET
ThrowOnBeforeExecute := _ThrowOnBeforeExecute;
END_GET
SET
_ThrowOnBeforeExecute := ThrowOnBeforeExecute;
END_SET
END_PROPERTY

END_FUNCTION_BLOCK

// ---- Tests/Automation/AutomationChildInitializationTimeoutTest.TcPOU
(*
SPDX-FileCopyrightText: © 2026 Oleksandr Tiutyk <trofimich@gmail.com>
SPDX-License-Identifier: MIT
License: https://opensource.org/license/mit
*)

(*!
<summary>Checks that an incomplete child enters INVALID after its initialization timeout.</summary>
<description>
Owns a fresh simulated automation fixture and advances one initialization call per PLC cycle.
The fixture limits attempts to fifty calls. No native resources or hardware are involved.
</description>
*)

{attribute 'no_assign'}
{attribute 'no_explicit_call' := 'do not call this function block directly'}
FUNCTION_BLOCK AutomationChildInitializationTimeoutTest EXTENDS TOF_Testing.MultiCycleTest
VAR_STAT
	{attribute 'hide'}
	_ClassName : STRING := __POUNAME();
END_VAR
VAR
	_Fixture : POINTER TO AutomationComponentTestFixture;
END_VAR

(*!
<summary>Creates the fixture, whose attempt limit bounds the scenario.</summary>
*)
METHOD PROTECTED BeforeTest
_Timeout := T#0S;
_Fixture := __NEW(AutomationComponentTestFixture);

IF _Fixture = 0 THEN
	TOF_Core.DynamicMemoryManager.RaiseAllocationFailure();
END_IF
END_METHOD

(*!
<summary>Advances one child initialization call and reports completion when the result is observable.</summary>
*)
METHOD PROTECTED ExecuteTest : TOF_Testing.TEST_CYCLE_RESULT
VAR
	assertions : REFERENCE TO TOF_Testing.Assertions;
END_VAR
assertions REF= Assert;
ExecuteTest := _Fixture^.AdvanceInitializationTimeout(assertions := assertions);
END_METHOD

(*!
<summary>Releases the fixture before publishing the result, after success or failure.</summary>
*)
METHOD PROTECTED AfterTest
VAR
	fixture : POINTER TO AutomationComponentTestFixture;
END_VAR
fixture := _Fixture;
_Fixture := 0;

IF fixture <> 0 THEN
	__DELETE(fixture);
END_IF
END_METHOD

(*!
<summary>Releases a still-owned fixture when the case is unloaded.</summary>
<param name="bInCopyCode">TwinCAT copy-code exit marker. Leave copied ownership with the new instance.</param>
*)
METHOD FB_exit : BOOL
VAR_INPUT
	bInCopyCode : BOOL;
END_VAR
IF NOT bInCopyCode AND_THEN _Fixture <> 0 THEN
	__DELETE(_Fixture);
END_IF

FB_exit := TRUE;
END_METHOD

(*!
<summary>Borrows the concrete class name. Callers must not modify it.</summary>
*)
{attribute 'monitoring' := 'call'}
PROPERTY ClassName : REFERENCE TO STRING
GET
ClassName REF= _ClassName;
END_GET
END_PROPERTY

(*!
<summary>Borrows the project namespace name. Callers must not modify it.</summary>
*)
{attribute 'monitoring' := 'call'}
PROPERTY NamespaceName : REFERENCE TO STRING
GET
NamespaceName REF= CurrentNamespace.Name;
END_GET
END_PROPERTY

(*!
<summary>Reports the complete instance size in bytes.</summary>
*)
{attribute 'monitoring' := 'call'}
PROPERTY SelfSize : ULINT
GET
SelfSize := XSIZEOF(THIS^);
END_GET
END_PROPERTY

END_FUNCTION_BLOCK

// ---- Tests/Automation/AutomationRunnerObservationTest.TcPOU
(*
SPDX-FileCopyrightText: © 2026 Oleksandr Tiutyk <trofimich@gmail.com>
SPDX-License-Identifier: MIT
License: https://opensource.org/license/mit
*)

(*!
<summary>Reports the selected result published by the dedicated automation runner test task.</summary>
<description>
Reads synchronized immutable diagnostics. A ten-second timer bounds the wait in the observing task.
Repeated runs re-read the publication. Reinitialize the application to execute the producer again.
</description>
*)

{attribute 'no_assign'}
{attribute 'no_explicit_call' := 'do not call this function block directly'}
FUNCTION_BLOCK AutomationRunnerObservationTest EXTENDS TOF_Testing.MultiCycleTest
VAR_STAT
	{attribute 'hide'}
	_ClassName : STRING := __POUNAME();
END_VAR
VAR CONSTANT
	//! <summary>Maximum real-time wait for publication.</summary>
	_PublicationTimeout : TIME := T#10S;
END_VAR
VAR
	_CheckInvalidRoots : BOOL;
	_Deadline : Tc2_Standard.TON;
END_VAR

(*!
<summary>Selects which published runner diagnostic this case reports.</summary>
<param name="name">Name reported for this case.</param>
<param name="parent">Group that owns this case.</param>
<param name="checkInvalidRoots">TRUE reads root validation. FALSE reads the normal execution result.</param>
*)
METHOD FB_init : BOOL
VAR_INPUT
	bInitRetains: BOOL; // TRUE: the retain variables are initialized (reset warm / reset cold)
	bInCopyCode: BOOL; // TRUE: the instance will be copied to the copy code afterward (online change)
	name : WSTRING;
	parent : TOF_Testing.ITestElement;
	checkInvalidRoots : BOOL;
END_VAR
IF NOT bInCopyCode THEN
	_CheckInvalidRoots := checkInvalidRoots;
END_IF

FB_init := TRUE;
END_METHOD

(*!
<summary>Clears the publication timer for a new runtime or Reset run.</summary>
*)
METHOD PROTECTED BeforeTest
_Timeout := T#0S;
_Deadline(IN := FALSE, PT := _PublicationTimeout);
END_METHOD

(*!
<summary>Polls synchronized publication once and reports the result when ready.</summary>
*)
METHOD PROTECTED ExecuteTest : TOF_Testing.TEST_CYCLE_RESULT
VAR
	happyPathFailure : STRING(255);
	invalidRootsFailure : STRING(255);
END_VAR
_Deadline(IN := TRUE, PT := _PublicationTimeout);
ExecuteTest := TOF_Testing.TEST_CYCLE_RESULT.DONE;

IF AutomationRunnerTestProgram.ReadResults(
	happyPathFailure => happyPathFailure,
	invalidRootsFailure => invalidRootsFailure
) THEN
	IF _CheckInvalidRoots THEN
		Assert.ThatString(actual := invalidRootsFailure, message := TO_WSTRING(invalidRootsFailure)).ToBe(expected := '');
	ELSE
		Assert.ThatString(actual := happyPathFailure, message := TO_WSTRING(happyPathFailure)).ToBe(expected := '');
	END_IF
ELSIF _Deadline.Q THEN
	RecordFailure(message := "RunnerTestTask did not publish within ten seconds");
ELSE
	ExecuteTest := TOF_Testing.TEST_CYCLE_RESULT.BUSY;
END_IF
END_METHOD

(*!
<summary>Borrows the concrete class name. Callers must not modify it.</summary>
*)
{attribute 'monitoring' := 'call'}
PROPERTY ClassName : REFERENCE TO STRING
GET
ClassName REF= _ClassName;
END_GET
END_PROPERTY

(*!
<summary>Borrows the project namespace name. Callers must not modify it.</summary>
*)
{attribute 'monitoring' := 'call'}
PROPERTY NamespaceName : REFERENCE TO STRING
GET
NamespaceName REF= CurrentNamespace.Name;
END_GET
END_PROPERTY

(*!
<summary>Reports the complete instance size in bytes.</summary>
*)
{attribute 'monitoring' := 'call'}
PROPERTY SelfSize : ULINT
GET
SelfSize := XSIZEOF(THIS^);
END_GET
END_PROPERTY

END_FUNCTION_BLOCK

